// TwinCAT 3 PLC project Controller
// Title: BIO2
// Company: 3P Innovation Ltd.
// Author: James Tyler
// ProgramVersion: 3.1.0.8
// libraries:
//   Standard, * (System)
//   Tc2_Standard, * (Beckhoff Automation GmbH)
//   Tc2_System, * (Beckhoff Automation GmbH)
//   Tc2_Utilities, * (Beckhoff Automation GmbH)
//   Tc2_XmlDataSrv, * (Beckhoff Automation GmbH)
//   Tc3_Interfaces, * (Beckhoff Automation GmbH)
//   Tc3_Module, * (Beckhoff Automation GmbH)
//   Tc_Persistent, * (Red Rock Controls Limited)
//   Tc2_MC2,newest,Beckhoff Automation GmbH
//   Tc_Collections,1.0.0.8,Red Rock Controls
//   Tc_Helper,1.0.0.8,Red Rock Controls
// project tree:
//   Classes/Compress/ FB_Compress.TcPOU
//   Classes/Config/ TConfig.TcPOU, TConfigData.TcDUT
//   Classes/Pusher/ FB_Pusher.TcPOU
//   Classes/Shield/ FB_Shield.TcPOU
//   DUTs/ st_language.TcDUT, St_Compress_Settings.TcDUT, E_LampState.TcDUT, E_CTRL_STATE.TcDUT (not stored), st_graph_visibility.TcDUT, Limits.TcDUT, Recipe.TcDUT (not stored), Rec_Compress.TcDUT, Rec_Other.TcDUT, Rec_Pusher.TcDUT, Rec_Clamp.TcDUT, Rec_Shield.TcDUT, st_recipe_titles.TcDUT, st_yellow_visibility.TcDUT
//   GVLs/ GVL_IO.TcGVL, GVL_Objects.TcGVL, GVL_ZenOn.TcGVL
//   / PlcTask.TcTTO, Task_Fast.TcTTO
//   POUs/ Config_Slow.TcPOU, FB_AxisControl.TcPOU, FB_LampController.TcPOU (not stored), F_DisplayText.TcPOU, PRG_MAIN.TcPOU, PRG_IO.TcPOU, PRG_Machine.TcPOU
//   XML/ eXMLState.TcDUT (not stored), FB_Retain.TcPOU (not stored), FB_RetainedData.TcPOU
// real-time tasks:
//   TASK PlcTask: cycle T#10ms, priority 12, ADS port 350
//   TASK Task_Fast: cycle T#1ms, priority 4, ADS port 351
// motion (NC):
//   TASK NC-Task 1 SAF: cycle T#2ms, priority 6, ADS port 501
//   TASK NC-Task 1 SVB: cycle T#10ms, priority 10, ADS port 511
//   AXIS Compress (id 1)
//     Dynamic: Acceleration=60.7875, Deceleration=60.7875, Jerk=182.363
//     Velo: RefSearch=0.40525, RefSync=0.40525, SlowManual=2.02625, FastManual=12.1575, Fast=40.525, Maximum=200
//     OtherSettings: AllowMotionCmdToSlave=true
//     encoder EncType=19
//       EncPara: ScaleFactorNumerator=0.5, ScaleFactorDenominator=1048576, ModuloFactor=0.5, MaxCount=#xffffffff
//     drive DrvType=16
//       DrvPara: MaxCount=#xffffffff
//         Analog: VeloReferenz=200, VeloScale=32
//         TimeComp: TaskDelayCycles=1
//     controller CtrType=1
//       CtrPara: PriorControlFactor=1
//         PosDiffControl: Enable=false, Range=0.05
//         PID: PosKp=20
//         Observer: BandWidth=20
//   AXIS Pusher (id 2)
//     Dynamic: Acceleration=60.7875, Deceleration=60.7875, Jerk=182.363
//     Velo: RefSearch=0.40525, RefSync=0.40525, SlowManual=2.02625, FastManual=12.1575, Fast=40.525, Maximum=40.525
//     OtherSettings: AllowMotionCmdToSlave=true
//     encoder EncType=19
//       EncPara: ScaleFactorNumerator=0.5, ScaleFactorDenominator=1048576, ModuloFactor=0.5, MaxCount=#xffffffff
//     drive DrvType=16
//       DrvPara: MaxCount=#xffffffff
//         Analog: VeloReferenz=100, VeloScale=32
//         TimeComp: TaskDelayCycles=1
//     controller CtrType=1
//       CtrPara: PriorControlFactor=1
//         PosDiffControl: Enable=false, Range=0.5
//         PID: PosKp=20
//         Observer: BandWidth=20
//   AXIS Shield (id 3)
//     Dynamic: Acceleration=60.7875, Deceleration=60.7875, Jerk=182.363
//     Velo: RefSearch=0.40525, RefSync=0.40525, SlowManual=2.02625, FastManual=12.1575, Fast=200, Maximum=200
//     OtherSettings: AllowMotionCmdToSlave=true
//     encoder EncType=19
//       EncPara: ScaleFactorNumerator=0.5, ScaleFactorDenominator=1048576, ModuloFactor=0.5, MaxCount=#xffffffff
//     drive DrvType=16
//       DrvPara: MaxCount=#xffffffff
//         Analog: VeloReferenz=200, VeloScale=32
//         TimeComp: TaskDelayCycles=1
//     controller CtrType=1
//       CtrPara: PriorControlFactor=1
//         PosDiffControl: Enable=false, Range=0.05
//         PID: PosKp=20
//         Observer: BandWidth=20
// I/O:
//   DEVICE Device 1 (EtherCAT), AmsNetId 5.49.191.228.2.1
//     Term 5 (EK1100) [EK1100 EtherCAT Coupler (2A E-Bus)]
//       Term 6 (EL1809) [EL1809 16Ch. Dig. Input 24V, 3ms]
//       Term 7 (EL2798) [EL2798 8Ch. Dig. Output 24V AC/DC, 2A, potential-free]
//       Term 13 (EL9011) [EL9011 End Terminal]
//     Term 8 (EK1100) [EK1100 EtherCAT Coupler (2A E-Bus)]
//       Term 9 (EL7201-9014) [EL7201-9014 1Ch. MDP742 Servo motor output stage with OCT (50V, 4A) and STO input]
//       Term 10 (EL7201-9014) [EL7201-9014 1Ch. MDP742 Servo motor output stage with OCT (50V, 4A)  and STO input]
//       Term 11 (EL7201-9014) [EL7201-9014 1Ch. MDP742 Servo motor output stage with OCT (50V, 4A)  and STO input]
//       Term 12 (EL1809) [EL1809 16Ch. Dig. Input 24V, 3ms]
//       Term 14 (EL9011) [EL9011 End Terminal]
//   DEVICE Device 3 (RT-Ethernet Protocol) (disabled), AmsNetId 5.49.191.228.4.1
// variable links:
//   NC-Task 1 SAF/Axes/Compress <-> Device 1 (EtherCAT)/Term 8 (EK1100)/Term 9 (EL7201-9014)
//     Drive/Inputs/In/nDcOutputTime <-> InfoData/DcOutputShift
//     Drive/Inputs/In/nState1 <-> DRV Statusword/Statusword
//     Drive/Inputs/In/nState2 <-> DRV Statusword/Statusword @bit 8
//     Drive/Inputs/In/nState4 @bit 1 <-> WcState/InputToggle
//     Drive/Inputs/In/nState4 <-> WcState/WcState
//     Drive/Outputs/Out/nCtrl1 <-> DRV Controlword/Controlword
//     Drive/Outputs/Out/nCtrl2 <-> DRV Controlword/Controlword @bit 8
//     Drive/Outputs/Out/nDataOut2 <-> DRV Target velocity/Target velocity
//     Enc/Inputs/In/nDataIn1 <-> FB Position/Position
//     Enc/Inputs/In/nDcInputTime <-> InfoData/DcInputShift
//     Enc/Inputs/In/nState4 @bit 1 <-> WcState/InputToggle
//     Enc/Inputs/In/nState4 <-> WcState/WcState
//   NC-Task 1 SAF/Axes/Pusher <-> Device 1 (EtherCAT)/Term 8 (EK1100)/Term 10 (EL7201-9014)
//     Drive/Inputs/In/nDcOutputTime <-> InfoData/DcOutputShift
//     Drive/Inputs/In/nState1 <-> DRV Statusword/Statusword
//     Drive/Inputs/In/nState2 <-> DRV Statusword/Statusword @bit 8
//     Drive/Inputs/In/nState4 @bit 1 <-> WcState/InputToggle
//     Drive/Inputs/In/nState4 <-> WcState/WcState
//     Drive/Outputs/Out/nCtrl1 <-> DRV Controlword/Controlword
//     Drive/Outputs/Out/nCtrl2 <-> DRV Controlword/Controlword @bit 8
//     Drive/Outputs/Out/nDataOut2 <-> DRV Target velocity/Target velocity
//     Enc/Inputs/In/nDataIn1 <-> FB Position/Position
//     Enc/Inputs/In/nDcInputTime <-> InfoData/DcInputShift
//     Enc/Inputs/In/nState4 @bit 1 <-> WcState/InputToggle
//     Enc/Inputs/In/nState4 <-> WcState/WcState
//   NC-Task 1 SAF/Axes/Shield <-> Device 1 (EtherCAT)/Term 8 (EK1100)/Term 11 (EL7201-9014)
//     Drive/Inputs/In/nDcOutputTime <-> InfoData/DcOutputShift
//     Drive/Inputs/In/nState1 <-> DRV Statusword/Statusword
//     Drive/Inputs/In/nState2 <-> DRV Statusword/Statusword @bit 8
//     Drive/Inputs/In/nState4 @bit 1 <-> WcState/InputToggle
//     Drive/Inputs/In/nState4 <-> WcState/WcState
//     Drive/Outputs/Out/nCtrl1 <-> DRV Controlword/Controlword
//     Drive/Outputs/Out/nCtrl2 <-> DRV Controlword/Controlword @bit 8
//     Drive/Outputs/Out/nDataOut2 <-> DRV Target velocity/Target velocity
//     Enc/Inputs/In/nDataIn1 <-> FB Position/Position
//     Enc/Inputs/In/nDcInputTime <-> InfoData/DcInputShift
//     Enc/Inputs/In/nState4 @bit 1 <-> WcState/InputToggle
//     Enc/Inputs/In/nState4 <-> WcState/WcState
//   Controller/Controller Instance <-> Device 1 (EtherCAT)/Term 5 (EK1100)/Term 6 (EL1809)
//     PlcTask Inputs/GVL_IO.ixCabinetE_StopButtonOkay <-> Channel 1/Cabinet E-Stop
//     PlcTask Inputs/GVL_IO.ixE_StopRelayOkay <-> Channel 2/Input
//     PlcTask Inputs/GVL_IO.ixGuardRelayOkay <-> Channel 3/Input
//     PlcTask Inputs/GVL_IO.ixResetButton <-> Channel 6/Input
//     PlcTask Inputs/GVL_IO.ixSpareIN4 <-> Channel 4/Input
//     PlcTask Inputs/GVL_IO.ixSpareIN5 <-> Channel 5/Input
//     PlcTask Inputs/GVL_IO.ixSpareIN7 <-> Channel 7/Input
//     PlcTask Inputs/GVL_IO.ixSpareIN8 <-> Channel 8/Input
//     PlcTask Inputs/GVL_IO.ixStartButton <-> Channel 9/Input
//     PlcTask Inputs/GVL_IO.ixStop_Button <-> Channel 10/Input
//   Controller/Controller Instance <-> Device 1 (EtherCAT)/Term 5 (EK1100)/Term 7 (EL2798)
//     PlcTask Outputs/GVL_IO.qxClamp <-> Channel 2/Output
//     PlcTask Outputs/GVL_IO.qxEnableE_Stop <-> Channel 1/Output
//     PlcTask Outputs/GVL_IO.qxResetButtonLamp <-> Channel 5/Output
//     PlcTask Outputs/GVL_IO.qxSpareOUT3 <-> Channel 3/Output
//     PlcTask Outputs/GVL_IO.qxStartButtonLamp <-> Channel 4/Output
//   Controller/Controller Instance <-> Device 1 (EtherCAT)/Term 8 (EK1100)/Term 10 (EL7201-9014)
//     PlcTask Inputs/GVL_IO.ibPusherServoTorque <-> DRV Torque actual value/Torque actual value
//   Controller/Controller Instance <-> Device 1 (EtherCAT)/Term 8 (EK1100)/Term 11 (EL7201-9014)
//     PlcTask Inputs/GVL_IO.ibShieldServoTorque <-> DRV Torque actual value/Torque actual value
//   Controller/Controller Instance <-> Device 1 (EtherCAT)/Term 8 (EK1100)/Term 12 (EL1809)
//     PlcTask Inputs/GVL_IO.ixCompressHomeSwitch <-> Channel 1/Input
//     PlcTask Inputs/GVL_IO.ixFanCartridgeDiagnostics <-> Channel 11/Input
//     PlcTask Inputs/GVL_IO.ixGuardOkay <-> Channel 9/Input
//     PlcTask Inputs/GVL_IO.ixMachineE_StopButtonOkay <-> Channel 10/Input
//     PlcTask Inputs/GVL_IO.ixPusherHomeSwitch <-> Channel 3/Input
//     PlcTask Inputs/GVL_IO.ixShieldHomeSwitch <-> Channel 5/Input
//     PlcTask Inputs/GVL_IO.ixStart_Button_Machine <-> Channel 7/Input
//   Controller/Controller Instance <-> Device 1 (EtherCAT)/Term 8 (EK1100)/Term 9 (EL7201-9014)
//     PlcTask Inputs/GVL_IO.ibCompressServoTorque <-> DRV Torque actual value/Torque actual value
//   Controller/Controller Instance <-> NC-Task 1 SAF/Axes/Compress
//     PlcTask Inputs/GVL_IO.CompressAxis.NcToPlc <-> Outputs/ToPlc
//     PlcTask Outputs/GVL_IO.CompressAxis.PlcToNc <-> Inputs/FromPlc
//   Controller/Controller Instance <-> NC-Task 1 SAF/Axes/Pusher
//     PlcTask Inputs/GVL_IO.PusherAxis.NcToPlc <-> Outputs/ToPlc
//     PlcTask Outputs/GVL_IO.PusherAxis.PlcToNc <-> Inputs/FromPlc
//   Controller/Controller Instance <-> NC-Task 1 SAF/Axes/Shield
//     PlcTask Inputs/GVL_IO.ShieldAxis.NcToPlc <-> Outputs/ToPlc
//     PlcTask Outputs/GVL_IO.ShieldAxis.PlcToNc <-> Inputs/FromPlc

CONFIGURATION Controller
    RESOURCE PLC ON TwinCAT3
        TASK PlcTask(INTERVAL := T#10ms, PRIORITY := 12);
        TASK Task_Fast(INTERVAL := T#1ms, PRIORITY := 4);
        PROGRAM PRG_MAIN WITH PlcTask : PRG_MAIN;
        PROGRAM Config_Slow WITH Task_Fast : Config_Slow;
    END_RESOURCE
END_CONFIGURATION

// ---- Classes/Config/TConfigData.TcDUT
{attribute 'pack_mode' := '0'}
TYPE TConfigData :
STRUCT
	
	//Limits
	con_max_limit_Compress 					:LREAL;
	con_max_limit_Shield 					:LREAL;
	con_max_limit_Pusher 					:LREAL;
	con_max_pusher_shield_diff				:LREAL;
	con_max_torque							:LREAL;
	
	//you are here
	//Rec1_Name        						:STRING;
	rec1_Name_1									:UDINT;
	rec1_Name_2									:UDINT;
	rec1_Name_3									:UDINT;
	rec1_Name_4									:UDINT;
	rec1_Name_5									:UDINT;
	
	rec1_Shield_Retract_Speed					:LREAL;
	rec1_Shield_Speed_1							:LREAL;
	rec1_Shield_Speed_2							:LREAL;
	rec1_Shield_Speed_3							:LREAL;
	rec1_Shield_Speed_4							:LREAL;
	rec1_Shield_Speed_5							:LREAL;
	rec1_Shield_Speed_6							:LREAL;
	rec1_Shield_Distance_1						:LREAL;
	rec1_Shield_Distance_2						:LREAL;
	rec1_Shield_Distance_3						:LREAL;
	rec1_shield_Distance_4						:LREAL;
	rec1_shield_Distance_5						:LREAL;
	rec1_shield_Distance_6						:LREAL;
	
	rec1_Compress_Initial_Speed					:LREAL;
	rec1_Compress_Initial_Distance				:LREAL;
	rec1_Compress_Relax_Distance					:LREAL;
	rec1_Compress_Retract_Speed					:LREAL;
	
	rec1_Pusher_Retract_Speed					:LREAL;
	rec1_Pusher_Speed_1							:LREAL;
	rec1_Pusher_Speed_2							:LREAL;
	rec1_Pusher_Speed_3							:LREAL;
	rec1_Pusher_Speed_4							:LREAL;
	rec1_Pusher_Speed_5							:LREAL;
	rec1_Pusher_Speed_6							:LREAL;
	rec1_Pusher_Distance_1						:LREAL;
	rec1_Pusher_Distance_2						:LREAL;
	rec1_Pusher_Distance_3						:LREAL;
	rec1_Pusher_Distance_4						:LREAL;
	rec1_Pusher_Distance_5						:LREAL;
	rec1_Pusher_Distance_6						:LREAL;
	
	rec1_Other_Compress_Home_Offset				:LREAL;
	rec1_Other_Pusher_Home_Offset				:LREAL;
	rec1_Other_Shield_Home_Offset				:LREAL;
	
	rec1_Clamp_Release_Instance					:LREAL;
	
	rec1_Memory_Free							:LREAL:=1;

	//Rec2_Name        						:STRING;
	rec2_Name_1									:UDINT;
	rec2_Name_2									:UDINT;
	rec2_Name_3									:UDINT;
	rec2_Name_4									:UDINT;
	rec2_Name_5									:UDINT;
	
	rec2_Shield_Retract_Speed					:LREAL;
	rec2_Shield_Speed_1							:LREAL;
	rec2_Shield_Speed_2							:LREAL;
	rec2_Shield_Speed_3							:LREAL;
	rec2_Shield_Speed_4							:LREAL;
	rec2_Shield_Speed_5							:LREAL;
	rec2_Shield_Speed_6							:LREAL;
	rec2_Shield_Distance_1						:LREAL;
	rec2_Shield_Distance_2						:LREAL;
	rec2_Shield_Distance_3						:LREAL;
	rec2_shield_Distance_4						:LREAL;
	rec2_shield_Distance_5						:LREAL;
	rec2_shield_Distance_6						:LREAL;
	
	rec2_Compress_Initial_Speed					:LREAL;
	rec2_Compress_Initial_Distance				:LREAL;
	rec2_Compress_Relax_Distance					:LREAL;
	rec2_Compress_Retract_Speed					:LREAL;
	
	rec2_Pusher_Retract_Speed					:LREAL;
	rec2_Pusher_Speed_1							:LREAL;
	rec2_Pusher_Speed_2							:LREAL;
	rec2_Pusher_Speed_3							:LREAL;
	rec2_Pusher_Speed_4							:LREAL;
	rec2_Pusher_Speed_5							:LREAL;
	rec2_Pusher_Speed_6							:LREAL;
	rec2_Pusher_Distance_1						:LREAL;
	rec2_Pusher_Distance_2						:LREAL;
	rec2_Pusher_Distance_3						:LREAL;
	rec2_Pusher_Distance_4						:LREAL;
	rec2_Pusher_Distance_5						:LREAL;
	rec2_Pusher_Distance_6						:LREAL;
	
	rec2_Other_Compress_Home_Offset				:LREAL;
	rec2_Other_Pusher_Home_Offset				:LREAL;
	rec2_Other_Shield_Home_Offset				:LREAL;
	
	rec2_Clamp_Release_Instance					:LREAL;
	
	rec2_Memory_Free							:LREAL:=1;

	//Rec3_Name        						:STRING;
	rec3_Name_1									:UDINT;
	rec3_Name_2									:UDINT;
	rec3_Name_3									:UDINT;
	rec3_Name_4									:UDINT;
	rec3_Name_5									:UDINT;
	
	rec3_Shield_Retract_Speed					:LREAL;
	rec3_Shield_Speed_1							:LREAL;
	rec3_Shield_Speed_2							:LREAL;
	rec3_Shield_Speed_3							:LREAL;
	rec3_Shield_Speed_4							:LREAL;
	rec3_Shield_Speed_5							:LREAL;
	rec3_Shield_Speed_6							:LREAL;
	rec3_Shield_Distance_1						:LREAL;
	rec3_Shield_Distance_2						:LREAL;
	rec3_Shield_Distance_3						:LREAL;
	rec3_shield_Distance_4						:LREAL;
	rec3_shield_Distance_5						:LREAL;
	rec3_shield_Distance_6						:LREAL;
	
	rec3_Compress_Initial_Speed					:LREAL;
	rec3_Compress_Initial_Distance				:LREAL;
	rec3_Compress_Relax_Distance					:LREAL;
	rec3_Compress_Retract_Speed					:LREAL;
	
	rec3_Pusher_Retract_Speed					:LREAL;
	rec3_Pusher_Speed_1							:LREAL;
	rec3_Pusher_Speed_2							:LREAL;
	rec3_Pusher_Speed_3							:LREAL;
	rec3_Pusher_Speed_4							:LREAL;
	rec3_Pusher_Speed_5							:LREAL;
	rec3_Pusher_Speed_6							:LREAL;
	rec3_Pusher_Distance_1						:LREAL;
	rec3_Pusher_Distance_2						:LREAL;
	rec3_Pusher_Distance_3						:LREAL;
	rec3_Pusher_Distance_4						:LREAL;
	rec3_Pusher_Distance_5						:LREAL;
	rec3_Pusher_Distance_6						:LREAL;
	
	rec3_Other_Compress_Home_Offset				:LREAL;
	rec3_Other_Pusher_Home_Offset				:LREAL;
	rec3_Other_Shield_Home_Offset				:LREAL;
	
	rec3_Clamp_Release_Instance					:LREAL;
	
	rec3_Memory_Free							:LREAL:=1;

	//Rec4_Name        						:STRING;
	rec4_Name_1									:UDINT;
	rec4_Name_2									:UDINT;
	rec4_Name_3									:UDINT;
	rec4_Name_4									:UDINT;
	rec4_Name_5									:UDINT;
	
	rec4_Shield_Retract_Speed					:LREAL;
	rec4_Shield_Speed_1							:LREAL;
	rec4_Shield_Speed_2							:LREAL;
	rec4_Shield_Speed_3							:LREAL;
	rec4_Shield_Speed_4							:LREAL;
	rec4_Shield_Speed_5							:LREAL;
	rec4_Shield_Speed_6							:LREAL;
	rec4_Shield_Distance_1						:LREAL;
	rec4_Shield_Distance_2						:LREAL;
	rec4_Shield_Distance_3						:LREAL;
	rec4_shield_Distance_4						:LREAL;
	rec4_shield_Distance_5						:LREAL;
	rec4_shield_Distance_6						:LREAL;
	
	rec4_Compress_Initial_Speed					:LREAL;
	rec4_Compress_Initial_Distance				:LREAL;
	rec4_Compress_Relax_Distance					:LREAL;
	rec4_Compress_Retract_Speed					:LREAL;
	
	rec4_Pusher_Retract_Speed					:LREAL;
	rec4_Pusher_Speed_1							:LREAL;
	rec4_Pusher_Speed_2							:LREAL;
	rec4_Pusher_Speed_3							:LREAL;
	rec4_Pusher_Speed_4							:LREAL;
	rec4_Pusher_Speed_5							:LREAL;
	rec4_Pusher_Speed_6							:LREAL;
	rec4_Pusher_Distance_1						:LREAL;
	rec4_Pusher_Distance_2						:LREAL;
	rec4_Pusher_Distance_3						:LREAL;
	rec4_Pusher_Distance_4						:LREAL;
	rec4_Pusher_Distance_5						:LREAL;
	rec4_Pusher_Distance_6						:LREAL;
	
	rec4_Other_Compress_Home_Offset				:LREAL;
	rec4_Other_Pusher_Home_Offset				:LREAL;
	rec4_Other_Shield_Home_Offset				:LREAL;
	
	rec4_Clamp_Release_Instance					:LREAL;

	rec4_Memory_Free							:LREAL:=1;		
	
	//Rec5_Name        						:STRING;
	rec5_Name_1									:UDINT;
	rec5_Name_2									:UDINT;
	rec5_Name_3									:UDINT;
	rec5_Name_4									:UDINT;
	rec5_Name_5									:UDINT;
	
	rec5_Shield_Retract_Speed					:LREAL;
	rec5_Shield_Speed_1							:LREAL;
	rec5_Shield_Speed_2							:LREAL;
	rec5_Shield_Speed_3							:LREAL;
	rec5_Shield_Speed_4							:LREAL;
	rec5_Shield_Speed_5							:LREAL;
	rec5_Shield_Speed_6							:LREAL;
	rec5_Shield_Distance_1						:LREAL;
	rec5_Shield_Distance_2						:LREAL;
	rec5_Shield_Distance_3						:LREAL;
	rec5_shield_Distance_4						:LREAL;
	rec5_shield_Distance_5						:LREAL;
	rec5_shield_Distance_6						:LREAL;
	
	rec5_Compress_Initial_Speed					:LREAL;
	rec5_Compress_Initial_Distance				:LREAL;
	rec5_Compress_Relax_Distance					:LREAL;
	rec5_Compress_Retract_Speed					:LREAL;
	
	rec5_Pusher_Retract_Speed					:LREAL;
	rec5_Pusher_Speed_1							:LREAL;
	rec5_Pusher_Speed_2							:LREAL;
	rec5_Pusher_Speed_3							:LREAL;
	rec5_Pusher_Speed_4							:LREAL;
	rec5_Pusher_Speed_5							:LREAL;
	rec5_Pusher_Speed_6							:LREAL;
	rec5_Pusher_Distance_1						:LREAL;
	rec5_Pusher_Distance_2						:LREAL;
	rec5_Pusher_Distance_3						:LREAL;
	rec5_Pusher_Distance_4						:LREAL;
	rec5_Pusher_Distance_5						:LREAL;
	rec5_Pusher_Distance_6						:LREAL;
	
	rec5_Other_Compress_Home_Offset				:LREAL;
	rec5_Other_Pusher_Home_Offset				:LREAL;
	rec5_Other_Shield_Home_Offset				:LREAL;
	
	rec5_Clamp_Release_Instance					:LREAL;
	
	rec5_Memory_Free							:LREAL:=1;
	
	//Rec6_Name        						:STRING;
	rec6_Name_1									:UDINT;
	rec6_Name_2									:UDINT;
	rec6_Name_3									:UDINT;
	rec6_Name_4									:UDINT;
	rec6_Name_5									:UDINT;
	
	rec6_Shield_Retract_Speed					:LREAL;
	rec6_Shield_Speed_1							:LREAL;
	rec6_Shield_Speed_2							:LREAL;
	rec6_Shield_Speed_3							:LREAL;
	rec6_Shield_Speed_4							:LREAL;
	rec6_Shield_Speed_5							:LREAL;
	rec6_Shield_Speed_6							:LREAL;
	rec6_Shield_Distance_1						:LREAL;
	rec6_Shield_Distance_2						:LREAL;
	rec6_Shield_Distance_3						:LREAL;
	rec6_shield_Distance_4						:LREAL;
	rec6_shield_Distance_5						:LREAL;
	rec6_shield_Distance_6						:LREAL;
	
	rec6_Compress_Initial_Speed					:LREAL;
	rec6_Compress_Initial_Distance				:LREAL;
	rec6_Compress_Relax_Distance					:LREAL;
	rec6_Compress_Retract_Speed					:LREAL;
	
	rec6_Pusher_Retract_Speed					:LREAL;
	rec6_Pusher_Speed_1							:LREAL;
	rec6_Pusher_Speed_2							:LREAL;
	rec6_Pusher_Speed_3							:LREAL;
	rec6_Pusher_Speed_4							:LREAL;
	rec6_Pusher_Speed_5							:LREAL;
	rec6_Pusher_Speed_6							:LREAL;
	rec6_Pusher_Distance_1						:LREAL;
	rec6_Pusher_Distance_2						:LREAL;
	rec6_Pusher_Distance_3						:LREAL;
	rec6_Pusher_Distance_4						:LREAL;
	rec6_Pusher_Distance_5						:LREAL;
	rec6_Pusher_Distance_6						:LREAL;
	
	rec6_Other_Compress_Home_Offset				:LREAL;
	rec6_Other_Pusher_Home_Offset				:LREAL;
	rec6_Other_Shield_Home_Offset				:LREAL;
	
	rec6_Clamp_Release_Instance					:LREAL;
	
	rec6_Memory_Free							:LREAL:=1;
	
	//Rec7_Name        						:STRING;
	rec7_Name_1									:UDINT;
	rec7_Name_2									:UDINT;
	rec7_Name_3									:UDINT;
	rec7_Name_4									:UDINT;
	rec7_Name_5									:UDINT;
	
	rec7_Shield_Retract_Speed					:LREAL;
	rec7_Shield_Speed_1							:LREAL;
	rec7_Shield_Speed_2							:LREAL;
	rec7_Shield_Speed_3							:LREAL;
	rec7_Shield_Speed_4							:LREAL;
	rec7_Shield_Speed_5							:LREAL;
	rec7_Shield_Speed_6							:LREAL;
	rec7_Shield_Distance_1						:LREAL;
	rec7_Shield_Distance_2						:LREAL;
	rec7_Shield_Distance_3						:LREAL;
	rec7_shield_Distance_4						:LREAL;
	rec7_shield_Distance_5						:LREAL;
	rec7_shield_Distance_6						:LREAL;
	
	rec7_Compress_Initial_Speed					:LREAL;
	rec7_Compress_Initial_Distance				:LREAL;
	rec7_Compress_Relax_Distance					:LREAL;
	rec7_Compress_Retract_Speed					:LREAL;
	
	rec7_Pusher_Retract_Speed					:LREAL;
	rec7_Pusher_Speed_1							:LREAL;
	rec7_Pusher_Speed_2							:LREAL;
	rec7_Pusher_Speed_3							:LREAL;
	rec7_Pusher_Speed_4							:LREAL;
	rec7_Pusher_Speed_5							:LREAL;
	rec7_Pusher_Speed_6							:LREAL;
	rec7_Pusher_Distance_1						:LREAL;
	rec7_Pusher_Distance_2						:LREAL;
	rec7_Pusher_Distance_3						:LREAL;
	rec7_Pusher_Distance_4						:LREAL;
	rec7_Pusher_Distance_5						:LREAL;
	rec7_Pusher_Distance_6						:LREAL;
	
	rec7_Other_Compress_Home_Offset				:LREAL;
	rec7_Other_Pusher_Home_Offset				:LREAL;
	rec7_Other_Shield_Home_Offset				:LREAL;
	
	rec7_Clamp_Release_Instance					:LREAL;
	
	rec7_Memory_Free							:LREAL:=1;
	
	//Rec8_Name        						:STRING;
	rec8_Name_1									:UDINT;
	rec8_Name_2									:UDINT;
	rec8_Name_3									:UDINT;
	rec8_Name_4									:UDINT;
	rec8_Name_5									:UDINT;
	
	rec8_Shield_Retract_Speed					:LREAL;
	rec8_Shield_Speed_1							:LREAL;
	rec8_Shield_Speed_2							:LREAL;
	rec8_Shield_Speed_3							:LREAL;
	rec8_Shield_Speed_4							:LREAL;
	rec8_Shield_Speed_5							:LREAL;
	rec8_Shield_Speed_6							:LREAL;
	rec8_Shield_Distance_1						:LREAL;
	rec8_Shield_Distance_2						:LREAL;
	rec8_Shield_Distance_3						:LREAL;
	rec8_shield_Distance_4						:LREAL;
	rec8_shield_Distance_5						:LREAL;
	rec8_shield_Distance_6						:LREAL;
	
	rec8_Compress_Initial_Speed					:LREAL;
	rec8_Compress_Initial_Distance				:LREAL;
	rec8_Compress_Relax_Distance					:LREAL;
	rec8_Compress_Retract_Speed					:LREAL;
	
	rec8_Pusher_Retract_Speed					:LREAL;
	rec8_Pusher_Speed_1							:LREAL;
	rec8_Pusher_Speed_2							:LREAL;
	rec8_Pusher_Speed_3							:LREAL;
	rec8_Pusher_Speed_4							:LREAL;
	rec8_Pusher_Speed_5							:LREAL;
	rec8_Pusher_Speed_6							:LREAL;
	rec8_Pusher_Distance_1						:LREAL;
	rec8_Pusher_Distance_2						:LREAL;
	rec8_Pusher_Distance_3						:LREAL;
	rec8_Pusher_Distance_4						:LREAL;
	rec8_Pusher_Distance_5						:LREAL;
	rec8_Pusher_Distance_6						:LREAL;
	
	rec8_Other_Compress_Home_Offset				:LREAL;
	rec8_Other_Pusher_Home_Offset				:LREAL;
	rec8_Other_Shield_Home_Offset				:LREAL;
	
	rec8_Clamp_Release_Instance					:LREAL;
	
	rec8_Memory_Free							:LREAL:=1;
	
	//Rec9_Name        						:STRING;
	rec9_Name_1									:UDINT;
	rec9_Name_2									:UDINT;
	rec9_Name_3									:UDINT;
	rec9_Name_4									:UDINT;
	rec9_Name_5									:UDINT;
	
	rec9_Shield_Retract_Speed					:LREAL;
	rec9_Shield_Speed_1							:LREAL;
	rec9_Shield_Speed_2							:LREAL;
	rec9_Shield_Speed_3							:LREAL;
	rec9_Shield_Speed_4							:LREAL;
	rec9_Shield_Speed_5							:LREAL;
	rec9_Shield_Speed_6							:LREAL;
	rec9_Shield_Distance_1						:LREAL;
	rec9_Shield_Distance_2						:LREAL;
	rec9_Shield_Distance_3						:LREAL;
	rec9_shield_Distance_4						:LREAL;
	rec9_shield_Distance_5						:LREAL;
	rec9_shield_Distance_6						:LREAL;
	
	rec9_Compress_Initial_Speed					:LREAL;
	rec9_Compress_Initial_Distance				:LREAL;
	rec9_Compress_Relax_Distance					:LREAL;
	rec9_Compress_Retract_Speed					:LREAL;
	
	rec9_Pusher_Retract_Speed					:LREAL;
	rec9_Pusher_Speed_1							:LREAL;
	rec9_Pusher_Speed_2							:LREAL;
	rec9_Pusher_Speed_3							:LREAL;
	rec9_Pusher_Speed_4							:LREAL;
	rec9_Pusher_Speed_5							:LREAL;
	rec9_Pusher_Speed_6							:LREAL;
	rec9_Pusher_Distance_1						:LREAL;
	rec9_Pusher_Distance_2						:LREAL;
	rec9_Pusher_Distance_3						:LREAL;
	rec9_Pusher_Distance_4						:LREAL;
	rec9_Pusher_Distance_5						:LREAL;
	rec9_Pusher_Distance_6						:LREAL;
	
	rec9_Other_Compress_Home_Offset				:LREAL;
	rec9_Other_Pusher_Home_Offset				:LREAL;
	rec9_Other_Shield_Home_Offset				:LREAL;
	
	rec9_Clamp_Release_Instance					:LREAL;
	
	rec9_Memory_Free							:LREAL:=1;
	
	//Rec10_Name        						:STRING;
	rec10_Name_1									:UDINT;
	rec10_Name_2									:UDINT;
	rec10_Name_3									:UDINT;
	rec10_Name_4									:UDINT;
	rec10_Name_5									:UDINT;
	
	rec10_Shield_Retract_Speed					:LREAL;
	rec10_Shield_Speed_1							:LREAL;
	rec10_Shield_Speed_2							:LREAL;
	rec10_Shield_Speed_3							:LREAL;
	rec10_Shield_Speed_4							:LREAL;
	rec10_Shield_Speed_5							:LREAL;
	rec10_Shield_Speed_6							:LREAL;
	rec10_Shield_Distance_1						:LREAL;
	rec10_Shield_Distance_2						:LREAL;
	rec10_Shield_Distance_3						:LREAL;
	rec10_shield_Distance_4						:LREAL;
	rec10_shield_Distance_5						:LREAL;
	rec10_shield_Distance_6						:LREAL;
	
	rec10_Compress_Initial_Speed					:LREAL;
	rec10_Compress_Initial_Distance				:LREAL;
	rec10_Compress_Relax_Distance					:LREAL;
	rec10_Compress_Retract_Speed					:LREAL;
	
	rec10_Pusher_Retract_Speed					:LREAL;
	rec10_Pusher_Speed_1							:LREAL;
	rec10_Pusher_Speed_2							:LREAL;
	rec10_Pusher_Speed_3							:LREAL;
	rec10_Pusher_Speed_4							:LREAL;
	rec10_Pusher_Speed_5							:LREAL;
	rec10_Pusher_Speed_6							:LREAL;
	rec10_Pusher_Distance_1						:LREAL;
	rec10_Pusher_Distance_2						:LREAL;
	rec10_Pusher_Distance_3						:LREAL;
	rec10_Pusher_Distance_4						:LREAL;
	rec10_Pusher_Distance_5						:LREAL;
	rec10_Pusher_Distance_6						:LREAL;
	
	rec10_Other_Compress_Home_Offset				:LREAL;
	rec10_Other_Pusher_Home_Offset				:LREAL;
	rec10_Other_Shield_Home_Offset				:LREAL;
	
	rec10_Clamp_Release_Instance					:LREAL;

	rec10_Memory_Free							:LREAL:=1;	
	
	(*Initialised - MUST BE LAST VARIABLE IN STUCTURE*)
    Initialised : BOOL;
END_STRUCT
END_TYPE

// ---- DUTs/st_language.TcDUT
TYPE st_language :
STRUCT
	portuguese				:BOOL:=FALSE;
	english					:BOOL:=TRUE;
END_STRUCT
END_TYPE

// ---- DUTs/St_Compress_Settings.TcDUT
TYPE St_Compress_Settings :
STRUCT
	
	//compress setting
	button					:BOOL;
	plus					:BOOL;
	minus					:BOOL;
	find					:BOOL;
	speed					:LREAL:=2;
	distance				:LREAL;
	old_distance			:LREAL;
	distance_vis			:BOOL;
	done					:BOOL;
	
END_STRUCT
END_TYPE

// ---- DUTs/E_LampState.TcDUT
TYPE E_LampState : 
(
	Off := 0,
    Steady := 1,
    FastFlash := 2,
    SlowFlash := 4
);
END_TYPE

// ---- DUTs/st_graph_visibility.TcDUT
TYPE st_graph_visibility :
	STRUCT
		shield_speed_1						:BOOL;
		shield_speed_2						:BOOL;
		shield_speed_3						:BOOL;
		shield_speed_4						:BOOL;
		shield_speed_5						:BOOL;
		shield_speed_6						:BOOL;
		shield_distance_1					:BOOL;
		shield_distance_2					:BOOL;
		shield_distance_3					:BOOL;
		shield_distance_4					:BOOL;
		shield_distance_5					:BOOL;
		shield_distance_6					:BOOL;
		shield_retract						:BOOL;
		
		pusher_speed_1						:BOOL;
		pusher_speed_2						:BOOL;
		pusher_speed_3						:BOOL;
		pusher_speed_4						:BOOL;
		pusher_speed_5						:BOOL;
		pusher_speed_6						:BOOL;
		pusher_distance_1					:BOOL;
		pusher_distance_2					:BOOL;
		pusher_distance_3					:BOOL;
		pusher_distance_4					:BOOL;
		pusher_distance_5					:BOOL;
		pusher_distance_6					:BOOL;
		pusher_retract						:BOOL;
		
		compress_initial_speed				:BOOL;
		compress_initial_distance			:BOOL;
		compress_relax_distance				:BOOL;
		compress_retract_speed				:BOOL;
	END_STRUCT
END_TYPE

// ---- DUTs/Limits.TcDUT
TYPE Limits :
	STRUCT
		max_limit_Compress				:LREAL;
		max_limit_Shield				:LREAL;
		max_limit_Pusher 				:LREAL;
		max_pusher_shield_diff			:LREAL;
		max_torque						:LREAL;
	END_STRUCT
END_TYPE

// ---- DUTs/Rec_Compress.TcDUT
TYPE Rec_Compress :
	STRUCT
		Initial_Speed				:LREAL;
		Initial_Distance			:LREAL;
		Relax_Distance				:LREAL;
		Retract_Speed				:LREAL;
	END_STRUCT
END_TYPE

// ---- DUTs/Rec_Other.TcDUT
TYPE Rec_Other :
	STRUCT
		Compress_Home_Offset		:LREAL;
		Pusher_Home_Offset			:LREAL;
		Shield_Home_Offset			:LREAL;

	END_STRUCT
END_TYPE

// ---- DUTs/Rec_Pusher.TcDUT
TYPE Rec_Pusher :
	STRUCT
		//Initial_Speed				:LREAL;
		//Initial_Distance			:LREAL;
		//Eject_Speed					:LREAL;
		//Eject_Distance				:LREAL;
		//Retract_Speed				:LREAL;
		//tamp_initial_speed			:LREAL;
		//tamp_final_speed			:LREAL;
		//tamp_initial_distance		:LREAL;
		//tamp_final_distance			:LREAL;
		
		Speed				:ARRAY[1..6] OF LREAL;
		Distance			:ARRAY[1..6] OF LREAL;
		retract_speed			:LREAL;
		
	END_STRUCT
END_TYPE

// ---- DUTs/Rec_Clamp.TcDUT
TYPE Rec_Clamp :
	STRUCT
		Release_Instance				:LREAL;
	END_STRUCT
END_TYPE

// ---- DUTs/Rec_Shield.TcDUT
TYPE Rec_Shield :
	STRUCT
		//Initial_Speed			:LREAL;
		//Initial_Distance		:LREAL;
		//Retract_Speed			:LREAL;
		Speed					:ARRAY[1..6] OF LREAL;
		Distance				:ARRAY[1..6] OF LREAL;
		retract_speed			:LREAL;
		
	END_STRUCT
END_TYPE

// ---- DUTs/st_recipe_titles.TcDUT
TYPE st_recipe_titles :
	STRUCT
		pusher					:STRING;
		compress				:STRING;
		shield					:STRING;
		clamp					:STRING;
		offset					:STRING;
		
	END_STRUCT
END_TYPE

// ---- DUTs/st_yellow_visibility.TcDUT
TYPE st_yellow_visibility :
STRUCT
	main				:BOOL;
	recipe				:BOOL;
	graph				:BOOL;
	maintenance			:BOOL;
	io					:BOOL;
	auto_mode			:BOOL;
	debug_mode			:BOOL;
END_STRUCT
END_TYPE

// ---- GVLs/GVL_IO.TcGVL
VAR_GLOBAL
	CompressAxis :AXIS_REF;	
	PusherAxis :AXIS_REF;	
	ShieldAxis :AXIS_REF;	
	ResetLampController : FB_LampController;
	StartLampController : FB_LampController;
	
	Name_String	AT%IB10 :STRING;
	Name_DINT1	AT%IB10	:DINT;
		
	// Cabinet Digital Inputs 1 - Device 1, Term 2
	ixCabinetE_StopButtonOkay AT%IX0.0 :BOOL;
	ixE_StopRelayOkay AT%IX0.1 :BOOL;
	ixGuardRelayOkay AT%IX0.2 :BOOL;
	ixSpareIN4 AT%IX0.3 :BOOL;
	ixSpareIN5 AT%IX0.4 :BOOL;
	ixResetButton AT%IX0.5 :BOOL;
	ixSpareIN7 AT%IX0.6 :BOOL;
	ixSpareIN8 AT%IX0.7 :BOOL;
	ixStart_Button_Machine AT%IX1.0 :BOOL;
	ixStop_Button AT%IX1.1 :BOOL;
	ixSpareIN11 AT%IX1.2 :BOOL;
	ixSpareIN12 AT%IX1.3 :BOOL;
	ixSpareIN13 AT%IX1.4 :BOOL;
	ixSpareIN14 AT%IX1.5 :BOOL;
	ixSpareIN15 AT%IX1.6 :BOOL;
	ixSpareIN16 AT%IX1.7 :BOOL;
	
	// Cabinet Digital Outputs 1 - Device 1, Term 3
	qxEnableE_Stop AT%QX0.0 :BOOL;
	qxClamp		 AT%QX0.1 :BOOL :=FALSE;
	qxSpareOUT3 AT%QX0.2 :BOOL;
	qxStartButtonLamp AT%QX0.3:BOOL;
	qxResetButtonLamp AT%QX0.4 :BOOL;
	qxSpareOUT6 AT%QX0.5 :BOOL;
	qxSpareOUT7 AT%QX0.6 :BOOL;
	qxSpareOUT8 AT%QX0.7 :BOOL;
	
	// Servo Analogue Inputs 1- Device 2, Term 2
	ibCompressServoTorque AT%IB120 :INT;
	ibCompressServoFollowingError AT%IB124 :DINT;
	qbCompressServoTorqueLimit AT%QB120 :UINT;
	
	// Servo Analogue Inputs 1- Device 2, Term 3
	ibPusherServoTorque AT%IB130 :INT;
	ibPusherServoFollowingError AT%IB134 :DINT;
	qbPusherServoTorqueLimit AT%QB130 :UINT;
	
	// Servo Analogue Inputs 1- Device 2, Term 3
	ibShieldServoTorque AT%IB140 :INT;
	ibShieldServoFollowingError AT%IB144 :DINT;
	qbShieldServoTorqueLimit AT%QB140 :UINT;
	
	// Analogue Inputs - Device 2, Term 4
	(*iiAnalogueIn7_HeaterTemperature AT%IB112 :INT;
	iiAnalogueIn8_UserProbeTemperature AT%IB114 :INT;
	// Status Inputs - Device 2, Term 4
	ixHeaterTC_Error AT%IX2.0 :BOOL;
	ixUserTC_Error AT%IX2.1 :BOOL;*)
	
	// Machine Digital Inputs 1 - Device 2, Term 5
	ixCompressHomeSwitch AT%IX2.0 :BOOL;
	ixPusherHomeSwitch AT%IX2.1 :BOOL;
	ixShieldHomeSwitch AT%IX2.2 :BOOL;
	ixStartButton AT%IX2.3 :BOOL;
	ixSpareIN25 AT%IX2.4 :BOOL;
	ixspareIN26 AT%IX2.5 :BOOL;
	ixspareIN27 AT%IX2.6 :BOOL;
	ixSpareIN28 AT%IX2.7 :BOOL;
	ixGuardOkay AT%IX3.0 :BOOL;
	ixMachineE_StopButtonOkay AT%IX3.1 :BOOL;
	ixFanCartridgeDiagnostics AT%IX3.2 :BOOL;
	ixSpareIN32 AT%IX3.3 :BOOL;
	ixSpareIN33 AT%IX3.4 :BOOL;
	ixSpareIN34 AT%IX3.5 :BOOL;
	ixSpareIN35 AT%IX3.6 :BOOL;
	ixSpareIN36 AT%IX3.7 :BOOL;

	CompressServoErrorID: UDINT;
	PusherServoErrorID: UDINT;	
	ShieldServoErrorID: UDINT;
	
	sSystemStateHi : STRING;
	sSystemStateMed : STRING;
	sSystemStateLo : STRING;
	
END_VAR

// ---- GVLs/GVL_Objects.TcGVL
VAR_GLOBAL
	Clock 						: TClock;
	Config 						: TConfig;
	configuring					: BOOL;
	config_request				: BOOL;
	Config_Message				: STRING(300);
	config_speed				: INT:=1;
	List_of_Recipes				: ARRAY[1..10] OF Recipe;
END_VAR

// ---- GVLs/GVL_ZenOn.TcGVL
VAR_GLOBAL
	
	//graph visibility
	graph_visibility							:st_graph_visibility;
	yellow_visibility							:st_yellow_visibility;
	yellow_visibility_old						:st_yellow_visibility;

	overtorque_alarm							:BOOL;

	limits_screen								:Limits;
	limits_save									:Limits;
	save_limits									:BOOL:=FALSE;
	parameter_violation							:BOOL:=FALSE;

	//Mode
	Debug_Mode									:BOOL;
	
	//Recipe on the screen (current one)
	Recipe_Visibility							:ARRAY[1..10] OF BOOL:=[10(FALSE)];  //u are here
	

	
	Recipe_Screen								:Recipe;
	Default_Recipe_Visibility					:BOOL :=FALSE;
		
	//end_of_recipe_on_the_screen
	
	//Maintenance
	Maintenance_Visibility						:BOOL;
	Mode_String									:STRING;
	Stage_Name									:STRING;
	Step_Next									:BOOL;
	Toggle_Clamp								:BOOL;
	Force_Home									:BOOL;
	//end of maintenance
	
	//recipe functions
	SaveRecipe									:BOOL :=FALSE;
	SaveasRecipe								:BOOL :=FALSE;	
	
	
	
	LoadRecipe									:ARRAY[1..10] OF BOOL :=[10(FALSE)];
	Load_Request								:BOOL :=FALSE;
	Save_before_load							:BOOL :=FALSE;
	
	DeleteRecipe								:ARRAY[1..10] OF BOOL :=[10(FALSE)];
	Delete_Request								:BOOL :=FALSE;
	
	

	Saveas_name									:STRING;
	Message										:STRING(300);
	alarm_message								:STRING(300);	
	question									:STRING(300);
	//current_recipe_message						:STRING;
	recipe_titles								:st_recipe_titles;
	language									:st_language;
	
	
	//end of recipe functions
	
	sc_CompressServoErrorID: UDINT;
	sc_PusherServoErrorID: UDINT;
	sc_ShieldServoErrorID: UDINT;
	sc_sSystemStateHi: STRING;
	sc_sSystemStateMed: STRING;
	sc_sSystemStateLo: STRING;
	

	
	// Servo Analogue Inputs 1- Device 2, Term 2
	CompressServoTorque          	: INT;
	CompressServoFollowingError		: DINT;
	CompressServoTorqueLimit		: UINT;
	
	// Servo Analogue Inputs 1- Device 2, Term 3
	PusherServoTorque				: INT;
	PusherServoFollowingError		: DINT;
	PusherServoTorqueLimit			: UINT;
	
	// Servo Analogue Inputs 1- Device 2, Term 3
	ShieldServoTorque				: INT;
	ShieldServoFollowingError		: DINT;
	ShieldServoTorqueLimit			: UINT;
		

	
	(* Data For the Main Screen *)
	//CurrentProcessState				: STRING;			//Main Screen

	

	
	(* Data For the Settings Screen *)
	//CompressDisplay					: LREAL;		//Settings Screen
	//PusherDisplay					: LREAL;		//Settings Screen
	//ShieldDisplay					: LREAL;
	
	Zenon_Offset_Compress			:BOOL;
	Zenon_Offset_Shield				:BOOL;
	Zenon_Offset_Pusher				:BOOL;
				
	
	(* Digital IO *)
	CabinetE_StopButtonOkay			: BOOL;
	E_StopRelayOkay					: BOOL;
	GuardRelayOkay					: BOOL;
	ResetButton                     : BOOL;
	EnableE_Stop					: BOOL;
	StartButtonLamp					: BOOL;
	ResetButtonLamp					: BOOL;
	
	Clamp_Alarm						:BOOL;
	Clamp_Cooling					:BOOL;
	Clamp_State						:BOOL;
	
	CompressHomeSwitch  			:BOOL;
	PusherHomeSwitch 				:BOOL;
	ShieldHomeSwitch 				:BOOL;
	StartButton 					:BOOL;

	GuardOkay 						:BOOL;
	MachineE_StopButtonOkay 		:BOOL;
	FanCartridgeDiagnostics 		:BOOL;

	ResetLamp						: BOOL;			//Digital IO Screen
	
	LampTest						: BOOL;			//Digital IO Screen

	CompressAxisPosition			: LREAL;		//IO Screen
	PusherAxisPosition				: LREAL;
	ShieldAxisPosition				: LREAL;
	
	//main
	product_count					: INT:=0;
	auto_cycle_time					: LREAL;
	actual_cycle_rate				: LREAL;
	
	compress_settings				:st_compress_settings;

END_VAR

// ---- POUs/PRG_MAIN.TcPOU
PROGRAM PRG_MAIN
VAR

	//test: BOOL;
	//debug: INT;
	all_config_initialised: BOOL;
	FirstScan			  : BOOL:=TRUE;
	temp: INT;
	arda: INT;
	bruce: INT;
END_VAR

//Recipes
Clock();


		
IF Config.Initialised() AND bruce < 70 THEN
	bruce:=bruce+1;
ELSIF Config.Initialised() THEN   
	arda := arda+1;
	PRG_IO();
	PRG_Machine();
END_IF

FirstSCan:=FALSE;

END_PROGRAM

// ---- POUs/PRG_IO.TcPOU
PROGRAM PRG_IO
VAR
	
	//piccirix		:INT;
	TextTimer: ton;
	Message_timer: ton;
	actual_cycle_timer: ton;
	

	recipe_default				:recipe;
	Current_Recipe				:Recipe;
	empty_recipe				:Recipe;
	current_recipe_no			:INT:=1;
	saveas_recipe_no			:INT;
	load_recipe_no				:INT;
	delete_recipe_no			:INT;
	temp						:INT;
	temp2						:INT;
		
	Initialise					:BOOL := TRUE;
	InitialiseTickCounter		:INT;
	TickCounter					:INT;
	
	save_requested				:BOOL;
	
	Pusher_Home					:BOOL;
	Shield_Home					:BOOL;
	Compress_Home				:BOOL;
	
	//violation
	//old_recipe					:Recipe;
	//old_limits					:Limits;
	zero_violation				:BOOL;
	max_distance_violation		:BOOL;
	max_sh_push_diff_violation	:BOOL;
	
	Message_old					:STRING(300);
	
	Message_State				:INT:=0;
	
	//deleting					:BOOL;
	//saving						:BOOL;
	//saving_as					:BOOL;
	//saving_lim					:BOOL;
	
	done						:BOOL:=FALSE;
	//you are here!!!!!!!!!!
	
	//cycles_waited				:INT;
	product_count_old			:INT;
	actual_cycle_array			: ARRAY[1..10] OF LREAL;
	
	
END_VAR

VAR_OUTPUT
					
END_VAR

ResetLampController();
StartLampController();
Message_timer();
actual_cycle_timer();

done:=TRUE;
//old_recipe:=current_recipe;
f_initialisation();

f_param_violation();

f_calc_auto_cycle_time();

f_calc_actual_cycle_rate();

f_alarms();

f_save_as();

f_load();

f_delete();

f_save();

f_save_limits();

f_configure_recipe();

f_titles();

f_message_timer();

//end recipes
f_leftbar_visibility();

f_digital_io();
		
f_mode_of_operation();

METHOD f_alarms : BOOL
VAR_INPUT
END_VAR
IF zero_violation THEN
	IF language.english THEN
		alarm_message:='Some parameters can not be set to zero.'; 
	ELSE
		alarm_message:='Alguns parâmetros não podem ser ajustados para zero.';
	END_IF
END_IF

IF max_distance_violation THEN
	
	IF language.english THEN
		alarm_message:='Maximum axis distance violation';
	ELSE
		alarm_message:='Violação máxima da distância do eixo';
	END_IF 
END_IF

IF max_sh_push_diff_violation THEN
	
	
	IF language.english THEN
		alarm_message:='Maximum pusher-shield distance difference violation';
	ELSE
		alarm_message:='Violação máxima da diferença de distância entre proteção-empurrador';
	END_IF 
 
END_IF

IF Clamp_Alarm THEN
	
	
	IF language.english THEN
		alarm_message:='Clamp Overtime';
	ELSE
		alarm_message:='Tempo adicional de grampo';
	END_IF 
END_IF

IF Overtorque_alarm THEN
	
	
	IF language.english THEN
		alarm_message:='Motor Overtorque';
	ELSE
		alarm_message:='Excesso de torque do motor';
	END_IF
	
END_IF

IF NOT ixGuardOkay THEN
	
	
	IF language.english THEN
		alarm_message:='Guard Open';
	ELSE
		alarm_message:='Guarda Aberto';
	END_IF
END_IF

IF NOT CabinetE_StopButtonOkay THEN
	
	IF language.english THEN
		alarm_message:='E-Stop Pressed';
	ELSE
		alarm_message:='Parada de emergência pressionada';
	END_IF
END_IF

IF CabinetE_StopButtonOkay AND ixGuardOkay AND NOT parameter_violation AND NOT Overtorque_alarm AND NOT Clamp_Alarm THEN
	alarm_message:='';
END_IF
END_METHOD

METHOD f_calc_actual_cycle_rate : BOOL
VAR
	cropped_product_count			:INT;
	temp_for						:INT;
	total_time						:LREAL;
END_VAR
actual_cycle_timer.IN:=TRUE;
actual_cycle_timer.PT:= T#604800S; //week



IF actual_cycle_timer.Q THEN
	//cycles_waited:=cycles_waited+1;
	actual_cycle_timer.IN:=FALSE;


ELSIF product_count_old <> product_count THEN
	
	actual_cycle_array[10]:=actual_cycle_array[9];
	actual_cycle_array[9]:=actual_cycle_array[8];
	actual_cycle_array[8]:=actual_cycle_array[7];
	actual_cycle_array[7]:=actual_cycle_array[6];
	actual_cycle_array[6]:=actual_cycle_array[5];
	actual_cycle_array[5]:=actual_cycle_array[4];
	actual_cycle_array[4]:=actual_cycle_array[3];
	actual_cycle_array[3]:=actual_cycle_array[2];
	actual_cycle_array[2]:=actual_cycle_array[1];
	
	
	actual_cycle_array[1]:=(*cycles_waited*300+*)TIME_TO_LREAL(actual_cycle_timer.ET);
	//cycles_waited:=0;
	actual_cycle_timer.IN:=FALSE;
	
	
END_IF


cropped_product_count:=product_count;

IF cropped_product_count > 10 THEN
	cropped_product_count:=10;
END_IF 

IF cropped_product_count <>0 THEN
	
	total_time:=0;
	FOR temp_for := 1 TO cropped_product_count DO
		total_time:=total_time+actual_cycle_array[temp_for];
	END_FOR
	
	actual_cycle_rate := ((cropped_product_count*3600000)/total_time);
	
ELSE
	total_time:=0;
	actual_cycle_rate:=0;
END_IF



product_count_old:=product_count;
END_METHOD

METHOD f_calc_auto_cycle_time : BOOL
VAR
	shield_time			:LREAL;
	pusher_time			:LREAL;
	compress_time		:LREAL;
	temp				:LREAL;
	temp_pusher			:LREAL;
	temp_shield			:LREAL;

	
	temp_for			:INT;
	
	auto_time_array		:ARRAY [1..8] OF LREAL;
	
END_VAR

compress_time := recipe_screen.Compress.Initial_Distance/recipe_screen.compress.Initial_Speed;
temp:=ABS(recipe_screen.Compress.Initial_Distance-recipe_screen.Compress.Relax_Distance);
compress_time := compress_time + (temp/recipe_screen.compress.Initial_Speed);         
auto_time_array[1] := compress_time;

temp_shield:=0;
temp_pusher:=0;

FOR temp_for := 2 TO 7 DO

	shield_time:=(ABS(recipe_screen.Shield.Distance[temp_for-1]-temp_shield))/recipe_screen.Shield.Speed[temp_for-1];
	temp_shield:=recipe_screen.Shield.Distance[temp_for-1];
	
	pusher_time:=(ABS(recipe_screen.Pusher.Distance[temp_for-1]-temp_pusher))/recipe_screen.Pusher.Speed[temp_for-1];
	temp_pusher:=recipe_screen.Pusher.Distance[temp_for-1];
	
	IF pusher_time > shield_time THEN
		auto_time_array[temp_for]:=pusher_time;	
	ELSE
		auto_time_array[temp_for]:=shield_time;
	END_IF
	
END_FOR

compress_time := recipe_screen.Compress.Relax_Distance/recipe_screen.Compress.Retract_speed;
shield_time := recipe_screen.Shield.Distance[6]/recipe_screen.Shield.retract_speed;
pusher_time := recipe_screen.Pusher.distance[6]/recipe_screen.pusher.retract_speed;

IF compress_time>=shield_time AND compress_time>=pusher_time THEN
	auto_time_array[8]:=compress_time;
END_IF

IF pusher_time>=shield_time AND pusher_time>=compress_time THEN
	auto_time_array[8]:=pusher_time;
END_IF

IF shield_time>=pusher_time AND shield_time>=compress_time THEN
	auto_time_array[8]:=shield_time;
END_IF

auto_cycle_time:=0;
FOR temp_for := 1 TO 8 DO
	auto_cycle_time:= auto_time_array[temp_for]+auto_cycle_time;
	
END_FOR
END_METHOD

METHOD f_configure_recipe : BOOL
VAR_INPUT
END_VAR

FOR temp := 1 TO 11 DO
	IF save_requested = TRUE THEN
		Config.CopyGlobalRecipiesToConfig();
		config_request:=TRUE;
		save_requested:=FALSE;
	END_IF
END_FOR
END_METHOD

METHOD f_delete : BOOL
VAR_INPUT
END_VAR
FOR temp := 1 TO 10 DO
	IF DeleteRecipe[temp] = TRUE THEN
		delete_recipe_no := temp;
		DeleteRecipe[temp] := FALSE;
		
		IF language.english THEN
			question := CONCAT('Do you want to delete recipe ', List_of_Recipes[delete_recipe_no].Name);
			question := CONCAT(question,'?');
		ELSE
			question := CONCAT('Deseja excluir a receita ', List_of_Recipes[delete_recipe_no].Name);
			question := CONCAT(question,'?');
		END_IF
 
	END_IF
END_FOR

IF Delete_Request = TRUE THEN
	
	Delete_Request:=FALSE;
	
	configuring:=TRUE;
	
	current_recipe_no:=delete_recipe_no;
	
	IF language.english THEN
		Message := CONCAT('Deleting recipe ',List_of_Recipes[current_recipe_no].Name );
		Message := CONCAT(Message,'...');

		Config_Message := concat('Recipe ', List_of_Recipes[current_recipe_no].Name);
		Config_Message := concat(Config_Message,' has been deleted.');
	ELSE
		Message := CONCAT('Excluindo receita ',List_of_Recipes[current_recipe_no].Name );
		Message := CONCAT(Message,'...');

		Config_Message := concat('A receita ', List_of_Recipes[current_recipe_no].Name);
		Config_Message := concat(Config_Message,' foi excluída.');
	END_IF
	
	WHILE (delete_recipe_no<10) AND List_of_Recipes[delete_recipe_no+1].Memory_Free = FALSE DO
		List_of_Recipes[delete_recipe_no]:=List_of_Recipes[delete_recipe_no+1];
		//save_requested[delete_recipe_no] := TRUE;
		delete_recipe_no:=delete_recipe_no+1;
	END_WHILE
	
	List_of_Recipes[delete_recipe_no] := empty_recipe;
	save_requested := TRUE;
	//List_of_Recipes[delete_recipe_no].Memory_Free:=FALSE;
	
	
	IF current_recipe_no = delete_recipe_no AND current_recipe_no <> 1 THEN
		current_recipe_no := current_recipe_no - 1;
	END_IF
		
	Current_Recipe := List_of_Recipes[current_recipe_no];
	recipe_screen:=current_recipe;
	
	
	
END_IF
END_METHOD

METHOD f_digital_io : BOOL
VAR_INPUT
END_VAR

(***************************** Data For the Main Screen ***********************)


CabinetE_StopButtonOkay := ixCabinetE_StopButtonOkay;
E_StopRelayOkay:=ixE_StopRelayOkay;
GuardRelayOkay:=ixGuardRelayOkay;
GuardOkay:=ixGuardOkay;

ResetButton := ixResetButton;

		
// Cabinet Digital Outputs 1 - Device 1, Term 3
EnableE_Stop:=qxEnableE_Stop;
	
//StartButtonLamp:=qxStartButtonLamp;
ResetButtonLamp:=qxResetButtonLamp;
	
	
// Servo Analogue Inputs 1- Device 2, Term 2
CompressServoTorque:=ibCompressServoTorque;
CompressServoFollowingError:=ibCompressServoFollowingError;
CompressServoTorqueLimit:=qbCompressServoTorqueLimit;
	
// Servo Analogue Inputs 1- Device 2, Term 3
PusherServoTorque:=ibPusherServoTorque;
PusherServoFollowingError:=ibPusherServoFollowingError;
PusherServoTorqueLimit:=qbPusherServoTorqueLimit;
	
// Servo Analogue Inputs 1- Device 2, Term 3
ShieldServoTorque:=ibShieldServoTorque;
ShieldServoFollowingError:=ibShieldServoFollowingError;
ShieldServoTorqueLimit:=qbShieldServoTorqueLimit;
	

	
// Machine Digital Inputs 1 - Device 2, Term 5
CompressHomeSwitch:=ixCompressHomeSwitch;
PusherHomeSwitch:=ixPusherHomeSwitch;
ShieldHomeSwitch:=ixShieldHomeSwitch;
StartButton:= ixStartButton;
GuardOkay:=ixGuardOkay; 
MachineE_StopButtonOkay:=ixMachineE_StopButtonOkay;
//FanCartridgeDiagnostics:=ixFanCartridgeDiagnostics;

//sc_CompressServoErrorID := CompressServoErrorID;
//sc_PusherServoErrorID := PusherServoErrorID;	
//sc_ShieldServoErrorID := ShieldServoErrorID;
	

//Homed?
Pusher_Home:=PRG_Machine.Pusher.HomeExecuted;
Shield_Home:=PRG_Machine.Shield.HomeExecuted;
Compress_Home:=PRG_Machine.Compress.HomeExecuted;
	
//Clamp
Clamp_State:=qxClamp;


qxResetButtonLamp := ResetLampController.Q; //io
ResetLamp := ResetLampController.Q; //zenon



ShieldAxisPosition := PRG_Machine.Shield.ShieldServo.fActualPosition;		
PusherAxisPosition := PRG_Machine.Pusher.PusherServo.fActualPosition;
CompressAxisPosition := PRG_Machine.Compress.CompressServo.fActualPosition;

Zenon_Offset_Compress:=PRG_Machine.Compress.OffsetExecuted;
Zenon_Offset_Shield:=PRG_Machine.Shield.OffsetExecuted;
Zenon_Offset_Pusher:=PRG_Machine.Pusher.OffsetExecuted;
END_METHOD

METHOD f_initialisation : BOOL
VAR
	//temp			:INT;
	
END_VAR

IF Initialise THEN
	//InitialiseTickCounter := InitialiseTickCounter + 1;
	//IF InitialiseTickCounter = 150 THEN
	//	Config.CopyConfigRecipiesToGlobal();
	//END_IF
	//piccirix:=piccirix+1;
	
	Config.CopyConfigRecipiesToGlobal();
		//piccirix:=piccirix+1;
	
	//piccirix:=piccirix+1;	
	//IF InitialiseTickCounter >= 300 THEN	
	//recipe_screen := List_of_Recipes[1];
	yellow_visibility.main:=TRUE;
	
	recipe_default.Name:='default 1';
	
	recipe_default.Compress.Initial_Distance:=5;
	recipe_default.Compress.Initial_Speed:=5;
	recipe_default.Compress.Relax_Distance:=3;
	recipe_default.Compress.Retract_Speed:=5;
	
	recipe_default.Pusher.Speed[1]:=5;
	recipe_default.Pusher.Speed[2]:=5;
	recipe_default.Pusher.Speed[3]:=5;
	recipe_default.Pusher.Speed[4]:=5;
	recipe_default.Pusher.Speed[5]:=5;
	recipe_default.Pusher.Speed[6]:=5;
	recipe_default.Pusher.Retract_Speed:=5;
	recipe_default.Pusher.Distance[1]:=5;
	recipe_default.Pusher.Distance[2]:=0;
	recipe_default.Pusher.Distance[3]:=5;
	recipe_default.Pusher.Distance[4]:=0;
	recipe_default.Pusher.Distance[5]:=5;
	recipe_default.Pusher.Distance[6]:=0;

	recipe_default.Shield.Speed[1]:=5;
	recipe_default.Shield.Speed[2]:=5;
	recipe_default.Shield.Speed[3]:=5;
	recipe_default.Shield.Speed[4]:=5;
	recipe_default.Shield.Speed[5]:=5;
	recipe_default.Shield.Speed[6]:=5;
	recipe_default.Shield.Retract_Speed:=5;
	recipe_default.Shield.Distance[1]:=5;
	recipe_default.Shield.Distance[2]:=0;
	recipe_default.Shield.Distance[3]:=5;
	recipe_default.Shield.Distance[4]:=0;
	recipe_default.Shield.Distance[5]:=5;
	recipe_default.Shield.Distance[6]:=0;
	
	recipe_default.Other.Compress_Home_Offset:=3;
	recipe_default.Other.Pusher_Home_Offset:=3;
	recipe_default.Other.Shield_Home_Offset:=3;
	
	recipe_default.Memory_Free:=FALSE;
	
	List_of_Recipes[1]:=recipe_default;
	recipe_screen:=List_of_Recipes[1];	
		
	limits_screen:=limits_save;
	
	IF language.english THEN
		Message:='Welcome!';
	ELSE
		Message:='Bem-vindo!';
	END_IF
	
	InitialiseTickCounter := 0;
	Initialise := FALSE;
	//END_IF		
ELSE
	//InitialiseTickCounter := 0;
	
	//FOR temp:=1 TO 11 DO
	///	Config.CopyConfigRecipiesToGlobal(temp);
		//piccirix:=piccirix+1;
	//END_FOR

	current_recipe:=recipe_screen;

	//current_recipe_message:=CONCAT('The current recipe number is ',INT_TO_STRING(Current_recipe_no));
	
	IF current_recipe_no = 1 THEN
		Default_Recipe_Visibility:=FALSE;
	ELSE
		Default_Recipe_Visibility:=TRUE;
	END_IF
	
	FOR	temp := 1 TO 10 DO
		Recipe_Visibility[temp]:=NOT(List_of_Recipes[temp].Memory_Free);
	END_FOR
	
	//temp:=1;
END_IF
END_METHOD

METHOD f_leftbar_visibility : BOOL
VAR_INPUT
END_VAR
IF NOT yellow_visibility_old.main AND yellow_visibility.main THEN
	yellow_visibility.recipe:=FALSE;
	yellow_visibility.maintenance:=FALSE;
	yellow_visibility.io:=FALSE;
	yellow_visibility.graph:=FALSE;
		
END_IF

IF NOT yellow_visibility_old.recipe AND yellow_visibility.recipe THEN
	yellow_visibility.main:=FALSE;
	yellow_visibility.maintenance:=FALSE;
	yellow_visibility.io:=FALSE;
	yellow_visibility.graph:=FALSE;
		
END_IF

IF NOT yellow_visibility_old.graph AND yellow_visibility.graph THEN
	yellow_visibility.main:=FALSE;
	yellow_visibility.maintenance:=FALSE;
	yellow_visibility.io:=FALSE;
	yellow_visibility.recipe:=FALSE;
		
END_IF

IF NOT yellow_visibility_old.io AND yellow_visibility.io THEN
	yellow_visibility.main:=FALSE;
	yellow_visibility.maintenance:=FALSE;
	yellow_visibility.graph:=FALSE;
	yellow_visibility.recipe:=FALSE;
		
END_IF

IF NOT yellow_visibility_old.maintenance AND yellow_visibility.maintenance THEN
	yellow_visibility.main:=FALSE;
	yellow_visibility.io:=FALSE;
	yellow_visibility.graph:=FALSE;
	yellow_visibility.recipe:=FALSE;
		
END_IF

yellow_visibility_old.main:=yellow_visibility.main;
yellow_visibility_old.maintenance:=yellow_visibility.maintenance;
yellow_visibility_old.recipe:=yellow_visibility.recipe;
yellow_visibility_old.graph:=yellow_visibility.graph;
yellow_visibility_old.io:=yellow_visibility.io;
END_METHOD

METHOD f_load : BOOL
VAR_INPUT
END_VAR
FOR temp := 1 TO 10 DO
	IF LoadRecipe[temp] = TRUE THEN
		load_recipe_no := temp;
		LoadRecipe[temp] := FALSE;
		

		
		IF language.english THEN
			question := CONCAT('Do you want to save recipe ', recipe_screen.Name);
			question := CONCAT(question,', before loading the recipe ');
			question := CONCAT(question, List_of_Recipes[load_recipe_no].Name);
			question := CONCAT(question,'?');			
		ELSE
			question := CONCAT('Deseja salvar a receita ', recipe_screen.Name);
			question := CONCAT(question,', antes de carregar a receita ');
			question := CONCAT(question, List_of_Recipes[load_recipe_no].Name);
			question := CONCAT(question,'?');			
		END_IF
 		
	END_IF
END_FOR

IF Load_Request = TRUE THEN
	
	Load_Request:=FALSE;
	
	IF(Save_before_load=TRUE)THEN
		
		configuring:=TRUE;
		//current_recipe:=recipe_screen;
		List_of_Recipes[current_recipe_no] := current_recipe;
		List_of_Recipes[current_recipe_no].Memory_Free := FALSE;
		//config.CopySettingsFromGlobal();
		Save_before_load := FALSE;
		
		IF language.english THEN
			Message := CONCAT('Saving recipe ',recipe_screen.Name);
			Message := CONCAT(Message,'... ');
		
			Config_Message := concat('Recipe ', recipe_screen.Name);
			Config_Message := concat(Config_Message,' has been saved.');
		ELSE
			
			Message := CONCAT('Salvando receita ',recipe_screen.Name);
			Message := CONCAT(Message,'... ');
		
			Config_Message := concat('A receita ', recipe_screen.Name);
			Config_Message := concat(Config_Message,' foi salva.');			
		END_IF
		save_requested := TRUE;	
		
	ELSE
		IF language.english THEN
			Message := CONCAT('Recipe ',List_of_Recipes[load_recipe_no].Name);
			Message := CONCAT(Message,' has been loaded');
		ELSE
			Message := CONCAT('A receita ',List_of_Recipes[load_recipe_no].Name);
			Message := CONCAT(Message,' foi carregada.');			
		END_IF
	END_IF
	
	current_recipe_no:=load_recipe_no;
		
	Current_Recipe := List_of_Recipes[current_recipe_no];
	recipe_screen:=current_recipe;
	//Message := CONCAT('Recipe ',current_recipe.Name);
	//Message := CONCAT(Message,' loading... ');

	
END_IF
END_METHOD

METHOD f_message_timer : BOOL
VAR_INPUT
END_VAR
CASE Message_State OF

0:
	
	IF Message <> message_old THEN
		//Message_State:=2;
		Message_timer.IN:=FALSE;
		Message_Timer.PT:=T#10S;
		Message_State:=0;
		
		Message_State:=1;
		
	END_IF
1:
	Message_timer.IN:=TRUE;
	Message_Timer.PT:=T#10S;
	Message_State:=0;
END_CASE

IF Message_Timer.Q = TRUE THEN
	Message:='';
	Message_timer.IN:=FALSE;
	Message_Timer.PT:=T#10S;
	//Message_Timer.PT:=T#30S;
END_IF 
Message_old:=Message;
END_METHOD

METHOD f_mode_of_operation : BOOL
VAR_INPUT
END_VAR
//Mode
IF debug_mode = FALSE THEN
	IF language.english THEN
		mode_string:= 'Current Mode: Automatic';
	ELSE
		mode_string:= 'Modo atual: Automático';
	END_IF
	yellow_visibility.auto_mode:=TRUE;
	yellow_visibility.debug_mode:=FALSE;
ELSE
	IF language.english THEN
		mode_string:= 'Current Mode: Debug';
	ELSE
		mode_string:= 'Modo atual: Depuração';
	END_IF
	yellow_visibility.auto_mode:=FALSE;
	yellow_visibility.debug_mode:=TRUE;
END_IF

//until here
END_METHOD

METHOD f_param_violation : BOOL
VAR
	pusher_calc				:ARRAY[0..6] OF LREAL;
	shield_calc				:ARRAY[0..6] OF LREAL;
	pusher_time				:LREAL;
	shield_time				:LREAL;
END_VAR
//violation

IF  
	recipe_screen.Compress.Initial_Speed =0 OR 
	recipe_screen.Compress.Retract_Speed =0 OR
	recipe_screen.pusher.speed[1] = 0 OR
	recipe_screen.pusher.speed[2] = 0 OR
	recipe_screen.pusher.speed[3] = 0 OR
	recipe_screen.pusher.speed[4] = 0 OR
	recipe_screen.pusher.speed[5] = 0 OR
	recipe_screen.pusher.speed[6] = 0 OR
	recipe_screen.Pusher.Retract_Speed = 0 OR
	recipe_screen.Shield.speed[1] = 0 OR
	recipe_screen.Shield.speed[2] = 0 OR
	recipe_screen.Shield.speed[3] = 0 OR
	recipe_screen.Shield.speed[4] = 0 OR
	recipe_screen.Shield.speed[5] = 0 OR
	recipe_screen.Shield.speed[6] = 0 OR
	recipe_screen.Shield.Retract_Speed = 0 THEN
		
	zero_violation := TRUE;
		
ELSE
	zero_violation := FALSE;
END_IF

IF 	recipe_screen.Other.Compress_Home_Offset > limits_screen.max_limit_compress OR
	recipe_screen.Other.Shield_Home_Offset > limits_screen.max_limit_Shield OR
	recipe_screen.Other.Pusher_Home_Offset > limits_screen.max_limit_Pusher OR
	
	recipe_screen.Compress.Initial_Distance + recipe_screen.Other.Compress_Home_Offset > limits_screen.max_limit_compress OR
	recipe_screen.Compress.Relax_Distance + recipe_screen.Other.Compress_Home_Offset > limits_screen.max_limit_compress OR
	
	recipe_screen.Shield.Distance[1] + recipe_screen.Other.shield_Home_Offset > limits_screen.max_limit_shield OR
	recipe_screen.Shield.Distance[2] + recipe_screen.Other.shield_Home_Offset > limits_screen.max_limit_shield OR
	recipe_screen.Shield.Distance[3] + recipe_screen.Other.shield_Home_Offset > limits_screen.max_limit_shield OR
	recipe_screen.Shield.Distance[4] + recipe_screen.Other.shield_Home_Offset > limits_screen.max_limit_shield OR
	recipe_screen.Shield.Distance[5] + recipe_screen.Other.shield_Home_Offset > limits_screen.max_limit_shield OR
	recipe_screen.Shield.Distance[6] + recipe_screen.Other.shield_Home_Offset > limits_screen.max_limit_shield OR
	
	recipe_screen.Pusher.Distance[1] + recipe_screen.Other.Pusher_Home_Offset > limits_screen.max_limit_pusher OR
	recipe_screen.Pusher.Distance[2] + recipe_screen.Other.Pusher_Home_Offset > limits_screen.max_limit_pusher OR
	recipe_screen.Pusher.Distance[3] + recipe_screen.Other.Pusher_Home_Offset > limits_screen.max_limit_pusher OR
	recipe_screen.Pusher.Distance[4] + recipe_screen.Other.Pusher_Home_Offset > limits_screen.max_limit_pusher OR
	recipe_screen.Pusher.Distance[5] + recipe_screen.Other.Pusher_Home_Offset > limits_screen.max_limit_pusher OR
	recipe_screen.Pusher.Distance[6] + recipe_screen.Other.Pusher_Home_Offset > limits_screen.max_limit_pusher THEN
	
	max_distance_violation:=TRUE;
	
ELSE
	max_distance_violation:=FALSE;
END_IF

max_sh_push_diff_violation := FALSE;

pusher_calc[0]:=recipe_screen.Other.Pusher_Home_Offset;
shield_calc[0]:=recipe_screen.Other.shield_Home_Offset;

FOR temp:=1 TO 6 DO
	pusher_calc[temp]:=recipe_screen.Other.Pusher_Home_Offset + recipe_screen.Pusher.Distance[temp];
	shield_calc[temp]:=recipe_screen.Other.Shield_Home_Offset + recipe_screen.Shield.Distance[temp];
END_FOR


FOR temp:=0 TO 6 DO
	IF pusher_calc[temp]-shield_calc[temp]> limits_screen.max_pusher_shield_diff THEN
		max_sh_push_diff_violation := TRUE;
	END_IF                         
END_FOR

FOR temp:=0 TO 5 DO
	pusher_time:=(pusher_calc[temp+1]-pusher_calc[temp])/recipe_screen.Pusher.Speed[temp+1];
	shield_time:=(shield_calc[temp+1]-shield_calc[temp])/recipe_screen.Shield.Speed[temp+1];
	IF recipe_screen.Pusher.Speed[temp+1] > recipe_screen.Shield.Speed[temp+1] AND pusher_time < shield_time THEN
    	IF pusher_calc[temp+1]-(pusher_time*recipe_screen.Shield.Speed[temp+1]+shield_calc[temp]) > limits_screen.max_pusher_shield_diff  THEN
			max_sh_push_diff_violation := TRUE;
		END_IF	
	
			
	END_IF                         
END_FOR


IF max_sh_push_diff_violation OR max_distance_violation OR zero_violation THEN
	parameter_violation:=TRUE;
ELSE
	parameter_violation:=FALSE;
END_IF


//violation end
END_METHOD

METHOD f_save : BOOL
VAR_INPUT
END_VAR
IF SaveRecipe THEN
	SaveRecipe := FALSE;

	current_recipe.Memory_Free:=FALSE;
	configuring:=TRUE;
	
	IF language.english THEN
		Message :=concat('Saving Recipe ',current_recipe.Name);	
		Message :=concat(Message,'...');
	
		Config_Message := concat('Recipe ', current_recipe.Name);
		Config_Message := concat(Config_Message,' has been saved.');
	ELSE
		Message :=concat('Salvando receita ',current_recipe.Name);	
		Message :=concat(Message,'...');
	
		Config_Message := concat('A receita ', current_recipe.Name);
		Config_Message := concat(Config_Message,' foi salva');
	END_IF
	
	List_of_Recipes[current_recipe_no] := current_recipe;
	save_requested := TRUE;
	
END_IF
END_METHOD

METHOD f_save_as : BOOL
VAR_INPUT
END_VAR
IF SaveasRecipe = TRUE THEN
	saveas_recipe_no:=current_recipe_no;
	WHILE (List_of_Recipes[saveas_recipe_no].Memory_Free = FALSE) AND (saveas_recipe_no<11) DO  
		saveas_recipe_no:=saveas_recipe_no+1;
		
	END_WHILE
	
	IF saveas_recipe_no > 10 THEN
		
		IF language.english THEN
			Message:='Maximum Recipe limit has been reached.';
		ELSE
			Message:='A limite máxima de receita foi alcançada.';
		END_IF
		
		saveas_recipe_no:=10;
		SaveasRecipe := FALSE;	
	
		
	ELSIF List_of_Recipes[saveas_recipe_no].Memory_Free = TRUE THEN
		SaveasRecipe:=FALSE;
		
		IF language.english THEN
			Message :=concat( 'Recipe ',current_recipe.Name);
			Message :=concat( Message,' is being saved as ');
			Message :=concat( Message,saveas_name);
			Message :=concat( Message,'...');
		
			Config_Message := concat('Recipe ', current_recipe.Name);
			Config_Message := concat(Config_Message,' has been saved as ');
			Config_Message := concat(Config_Message,saveas_name);
			Config_Message := concat(Config_Message,'.');
		ELSE //ure here........
			Message :=concat( 'A receita ',current_recipe.Name);
			Message :=concat( Message,' está sendo salva como ');
			Message :=concat( Message,saveas_name);
			Message :=concat( Message,'...');
		
			Config_Message := concat('A receita ', current_recipe.Name);
			Config_Message := concat(Config_Message,' foi salva como receita ');
			Config_Message := concat(Config_Message,saveas_name);
			Config_Message := concat(Config_Message,'.');			
		END_IF
		
		configuring:=TRUE;
		save_requested := TRUE;

		List_of_Recipes[saveas_recipe_no]:=current_recipe;
		List_of_Recipes[saveas_recipe_no].Name:=Saveas_name;
		List_of_Recipes[saveas_recipe_no].Memory_Free:=FALSE;
		//current_recipe:=recipe_screen;
		//Config.CopyGlobalRecipiesToConfig();
		
		//Current_Recipe := List_of_Recipes[current_recipe_no];
		//recipe_screen:=current_recipe;

				
	
	END_IF
	
END_IF
END_METHOD

METHOD f_save_limits : BOOL
VAR_INPUT
END_VAR
IF save_limits THEN
	save_limits:=FALSE;
	limits_save:=limits_screen;
	save_requested := TRUE;
	
	IF language.english THEN
		Message:='Saving Limits...';
	ELSE
		Message:='Salvando limites...';
	END_IF
		
	Config_Message:='Limits has been saved';
	configuring:=TRUE;
END_IF
END_METHOD

METHOD f_titles : BOOL
VAR_INPUT
END_VAR

IF language.english THEN
	recipe_titles.clamp:=concat( 'Clamp parameters for recipe ',recipe_screen.Name); 
	recipe_titles.clamp:=concat( recipe_titles.clamp,':');
ELSE
	recipe_titles.clamp:=concat( 'Parâmetros do grampo para receita ',recipe_screen.Name); 
	recipe_titles.clamp:=concat( recipe_titles.clamp,':');
END_IF

IF language.english THEN
	recipe_titles.compress:=concat( 'Compress parameters for recipe ',recipe_screen.Name); 
	recipe_titles.compress:=concat( recipe_titles.compress,':');
ELSE
	recipe_titles.compress:=concat( 'Parâmetros de compressão para receita ',recipe_screen.Name); 
	recipe_titles.compress:=concat( recipe_titles.compress,':');	
END_IF

IF language.english THEN
	recipe_titles.offset:=concat( 'Offset parameters for recipe receita ',recipe_screen.Name); 
	recipe_titles.offset:=concat( recipe_titles.offset,':');
ELSE
	recipe_titles.offset:=concat( 'Parâmetros de desvio para receita ',recipe_screen.Name); 
	recipe_titles.offset:=concat( recipe_titles.offset,':');
END_IF

IF language.english THEN
	recipe_titles.shield:=concat( 'Shield parameters for recipe ',recipe_screen.Name); 
	recipe_titles.shield:=concat( recipe_titles.shield,':');
ELSE
	recipe_titles.shield:=concat( 'Parâmetros de proteção para receita ',recipe_screen.Name); 
	recipe_titles.shield:=concat( recipe_titles.shield,':');
END_IF

IF language.english THEN
	recipe_titles.pusher:=concat( 'Pusher parameters for recipe ',recipe_screen.Name); 
	recipe_titles.pusher:=concat( recipe_titles.pusher,':');
ELSE
	recipe_titles.pusher:=concat( 'Parâmetros do empurrador para receita ',recipe_screen.Name); 
	recipe_titles.pusher:=concat( recipe_titles.pusher,':');
END_IF
END_METHOD

END_PROGRAM

// ---- POUs/PRG_Machine.TcPOU
PROGRAM PRG_Machine
VAR
	
	//empty recipe
	empty_recipe				:recipe;
	
	//debug
	after_debug_state					:INT :=0;

	
	Pusher :FB_Pusher;
	Compress: FB_Compress;
	Shield: FB_Shield;

	ZenonStart: NT_StartProcess;

	
	debug_counter: INT;
	tickcounter: INT;
	tickcounter2: INT;

	State: INT:= 0;
	state_old: INT:=0;
	StateNext: INT:= 0;
	
	SM_StepRequest: BOOL:=FALSE;
	singleStep: BOOL:=FALSE;
		
	Clamp_Security_Time: TIME := T#30S;
	ClampTimer: TON;
	//DwellTimer: TON;
	//SaveTickCounter: INT := 0;

	DatumTaught: BOOL;

	

	
	//stage
	stage_sh_push						:INT:=1;
	
END_VAR

VAR_OUTPUT

	rec_old		:recipe;
END_VAR

IF TRUE THEN
	debug_counter := debug_counter+1;
END_IF



qbCompressServoTorqueLimit := 1000;
qbPusherServoTorqueLimit := 1000;
qbShieldServoTorqueLimit := 1000;


//The state-machine
CASE State OF
	
0: //Copy config .txt file into machine settings
	


	//Zenon start process function call - appears to never generate errors
	
	//IF ZenonStart.Busy=FALSE THEN
	ZenonStart (
		NETID :=,
		//PATHSTR := 'Hard Disk\CP6606_Runtime\zenonRCE.exe', //'C:\PROGRAM Files\COPA-DATA\zenon 7.20 SP0\Zenrt32.exe',
		//DIRNAME := 'Hard Disk\CP6606_Runtime',  //'C:\Program Files\COPA-DATA\zenon 7.20 SP0',
		PATHSTR := 'Hard Disk\ZenonRunTime\zenonRCE.exe', //'C:\PROGRAM Files\COPA-DATA\zenon 7.20 SP0\Zenrt32.exe',
		DIRNAME := 'Hard Disk\ZenonRunTime',  //'C:\Program Files\COPA-DATA\zenon 7.20 SP0',
		COMNDLINE := '',
		START := TRUE,
		TMOUT := DEFAULT_ADS_TIMEOUT
		);
	StateNext := 10;



10: 
	qxEnableE_Stop := FALSE;
	tickcounter := 0;
	StateNext := 15;

15: //Check E-Stop relay is not set then Enable and initialise stuff - disable drive to clear errors

	

	//IF ixCabinetE_StopButtonOkay THEN
	qxEnableE_Stop := TRUE;
	StateNext := 20;
	//ELSE
	//	ResetLampController.State := SlowFlash;
	//END_IF
	
20: // Look for E-Stop button reset
	IF ixCabinetE_StopButtonOkay THEN
		//ResetLampController.State := steady;
		StateNext := 30;
	ELSE
		 
		ResetLampController.State := SlowFlash;
			
	END_IF
	
	//here
30: // Wait for operator to hit reset button
	
	IF ixE_StopRelayOkay THEN
		ResetLampController.State := off;
		StateNext := 40;
		tickcounter := 0;
	ELSE
		ResetLampController.State := steady;
		


	END_IF

40: // look for guard closed - disable drive to clear errors
	//sSystemStateMed := F_DisplayText("Guard Open",0);	
	//CurrentProcessState	:= F_DisplayText("not ready",0);	//Main Screen	

	
	IF NOT ixGuardOkay THEN
		ResetLampController.State := FastFlash;		
	ELSE
		ResetLampController.State := off;
		//sSystemStateMed := F_DisplayText("Initialising Axes",0);	
		tickcounter := 0;
		StateNext := 50;
	END_IF

50:
	IF ixGuardRelayOkay THEN
		statenext:=100;
	END_IF
	
100: // wait 2 scans for power supply to drive to stabilise
	tickcounter := tickcounter + 1;
	IF tickcounter >= 2 THEN
		tickcounter := 0;
		StateNext := 105;
	END_IF

105:
	IF NOT ixresetbutton THEN
		statenext:=110;
	END_IF	
	
110: // prepare for Servo motion - enable drive
//you are here!!!!!!!!!!!!!!!!!!!!!!!!!!!!
	//IF NOT ixResetButton THEN
		
		
	
	Shield._Enable();
	Pusher._Enable();
	Compress._Enable();
		
	tickcounter := tickcounter + 1;
	IF tickcounter >= 100 THEN
		tickcounter := 0;

		StateNext := 115;
	END_IF	
	//END_IF


	
115: 
	
	//IF Shield.HomeExecuted = FALSE OR Pusher.HomeExecuted = FALSE OR Compress.HomeExecuted = FALSE THEN
	IF language.english THEN
		Stage_Name := 'Beginning';
	ELSE
		Stage_Name := 'Início';
	END_IF
	Maintenance_Visibility:=TRUE;
	qxStartButtonLamp:=TRUE;
	IF (ixStartButton OR Step_Next OR ixStart_Button_Machine) THEN
		IF (parameter_violation = FALSE) THEN
			qxStartButtonLamp:=FALSE;
			StateNext := 116;
			Step_Next := FALSE;
			Clamp_Alarm:=FALSE;
			Maintenance_Visibility:=FALSE;
			stage_sh_push:=1;
			//Stage_Name := 'Homing and Offsetting';



		ELSE
			Step_Next:=FALSE;
		END_IF
	END_IF

	
116:
	IF (NOT ixstartbutton) AND NOT ixstart_button_machine THEN
		//general_offset_update();

		
		statenext:=117;
	END_IF
	
117:
	IF Compress.HomeExecuted=TRUE AND 
	   Shield.HomeExecuted = TRUE AND 
	   Pusher.HomeExecuted = TRUE AND
	   Pusher.OffsetExecuted = TRUE AND
	   Shield.OffsetExecuted = TRUE AND
	   Compress.OffsetExecuted = TRUE AND
	   Debug_Mode = FALSE THEN
	   
	   statenext:= 130;
	ELSE
		statenext:=120;
	END_IF
	
	Shield.Shield_param:=recipe_screen;
	Compress.Compress_Param := recipe_screen;
	Pusher.Pusher_Param := recipe_screen;
	//ELSE
	//	StateNext:=129;
	//	after_debug_state:=128;
	//END_IF
		
120: //you are here!!!!!!!!!!!!

	IF language.english THEN
		Stage_Name := 'Homing';
	ELSE
		Stage_Name := 'Ir para Início';
	END_IF
	IF Pusher.HomeExecuted = FALSE THEN 
		Pusher._Home();
	END_IF
	
	IF Compress.HomeExecuted = FALSE THEN
		Compress._Home();
	END_IF
	
	
	IF Compress.HomeExecuted AND Pusher.HomeExecuted THEN
		StateNext := 125;                //directly to end
		//Compress.HomeExecuted:=FALSE;
		//Pusher.HomeExecuted:=FALSE;
		
	END_IF
	
125:
	//random:='arda';
	IF Shield.HomeExecuted = FALSE THEN
		Shield._Home();
		
	ELSE
		StateNext := 129;
		IF language.english THEN
			Stage_Name := 'Homing done';
		ELSE
			Stage_Name := 'Ir para início concluído';
		END_IF
		after_debug_state :=127;
		//Shield.HomeExecuted := FALSE;
	END_IF

127:
	
	IF language.english THEN	
		Stage_Name := 'Offsetting';
	ELSE
		Stage_Name := 'Desviando';
	END_IF
	
	IF Compress.OffsetExecuted = FALSE THEN
		Compress.Offset(enable:=TRUE);
	END_IF
	
	IF Shield.OffsetExecuted = FALSE THEN
		Shield.Offset(enable:=TRUE);
	END_IF
	
	IF Pusher.OffsetExecuted = FALSE THEN
		Pusher.Offset(enable:=TRUE);
	END_IF
	
	IF Pusher.OffsetExecuted AND Shield.OffsetExecuted AND Compress.OffsetExecuted THEN
		Pusher.Offset(enable:=FALSE);
		Shield.Offset(enable:=FALSE);
		Compress.Offset(enable:=FALSE);
		
		rec_old:=Shield.Shield_Param;     //old values
		
		IF language.english THEN
			Stage_Name := 'Offsetting done';
		ELSE
			Stage_Name :='Desvio concluído';	
		END_IF
		
		Maintenance_Visibility := TRUE;
		qxStartButtonLamp:=TRUE;
		IF (ixStartButton OR Step_Next OR ixStart_Button_Machine) THEN
			IF (parameter_violation =FALSE) THEN
				qxStartButtonLamp:=FALSE;
				
				Shield.Shield_param:=recipe_screen;
				Compress.Compress_Param := recipe_screen;
				Pusher.Pusher_Param := recipe_screen;
			
				StateNext:=128;
				Step_Next:=FALSE;
				Maintenance_Visibility := FALSE;
			ELSE
				Step_Next:=FALSE;
			END_IF
		END_IF
	END_IF
	
128:	
	IF NOT ixstartbutton AND NOT ixstart_button_machine THEN
		statenext:=130;
	END_IF	

129: //debug	
	
	IF _debug(enable:=TRUE) THEN
		_debug(enable:=FALSE);
		statenext:=131;
	END_IF
		
130: //stage 1

	//IF ixstartbutton AND NOT ixstart_button_machine THEN
	IF language.english THEN
		Stage_Name := 'Compress Tobacco';
	ELSE
		Stage_Name := 'Comprimir Tabaco';
	END_IF
	
	IF qxClamp = FALSE THEN
		qxClamp:=TRUE;
		ClampTimer.IN:=TRUE;
		ClampTimer.PT:=Clamp_Security_Time;

	END_IF
	
	//IF Compress.Stage1Executed = FALSE THEN

	Compress._compress_tobacco(Enable:=TRUE);
	Compress.HomeExecuted:=FALSE;	
	
	IF Compress.axis_ready THEN	//Compress.Stage1Executed := FALSE;
		StateNext := 129;
		after_debug_state:=135;
		Compress._compress_tobacco(Enable:=FALSE);
		
		
		IF language.english THEN
			Stage_Name := 'Compress Tobacco done';
		ELSE
			Stage_Name := 'Comprimir tabaco concluído';
		END_IF
		
	END_IF
	//END_IF

131: //after_each_debug
	IF NOT ixStartButton AND NOT ixStart_Button_Machine THEN
	
		statenext:=after_debug_state;
	END_IF
135://stage2
	
	IF language.english THEN
		Stage_Name := concat('Shield-Pusher Stage ',INT_TO_STRING(stage_sh_push));
	ELSE
		Stage_Name := concat('Empurrador-proteção Estágio',INT_TO_STRING(stage_sh_push));
	END_IF
	
	Pusher.HomeExecuted:=FALSE;
	Shield.HomeExecuted:=FALSE;
		
	Pusher._absolute_move(Enable:=TRUE,Stage:=stage_sh_push);
	Shield._absolute_move(Enable:=TRUE,Stage:=stage_sh_push);
	IF pusher.axis_ready AND shield.axis_ready THEN	
		Statenext:= 129;
		IF stage_sh_push =6 THEN
			after_debug_state := 150;
			stage_sh_push:=0;
		ELSE
			after_debug_state := 135;
		END_IF
		Pusher._absolute_move(Enable:=FALSE,Stage:=stage_sh_push);
		Shield._absolute_move(Enable:=FALSE,Stage:=stage_sh_push);
		stage_sh_push:=stage_sh_push+1;
		
		IF language.english THEN
			Stage_Name:=concat(Stage_Name,' done');
		ELSE
			Stage_Name:=concat(Stage_Name,' concluído');
		END_IF
	END_IF	
	


150: //stage 5
	IF language.english THEN
		Stage_Name := 'Retract all';
	ELSE
		Stage_Name := 'Retrair tudo';
	END_IF
	//IF 	Shield._retract(Enable:=TRUE) AND Pusher._retract(Enable:=TRUE) AND Compress._retract(Enable:=TRRUE) THEN
	Pusher._Retract(enable:=TRUE);
	Shield._retract(enable:=TRUE);
	Compress._retract(enable:=TRUE);

	IF Compress.axis_ready AND Shield.Axis_ready AND Pusher.axis_ready THEN
		Pusher._Retract(enable:=FALSE);
		Shield._retract(enable:=FALSE);
		Compress._retract(enable:=FALSE);
		Statenext:=290;
		
		IF language.english THEN
			Stage_Name := 'Retract All Done';
		ELSE
			Stage_Name := 'Retrair tudo concluído';
		END_IF
	END_IF	

290:
	product_count:=product_count+1;
	statenext:=300;


300: //end
	
	Pusher.HomeExecuted:= TRUE;
	Shield.HomeExecuted:=TRUE;
	Compress.HomeExecuted:=TRUE;
	statenext:= 115;

	
1000: // overtorque
	
	//StartLoad := FALSE;
	
	tickcounter:=0;
	
	qxclamp:=FALSE;
	ClampTimer.IN:=FALSE;
	ClampTimer.PT:=Clamp_Security_Time;
	
	IF Pusher.PusherServo.xstopped AND Shield.ShieldServo.xstopped AND Compress.CompressServo.xstopped THEN
		Pusher._Reset();
		Shield._Reset();
		Compress._Reset();
		Statenext:=1005;
	END_IF

1005:
	
	IF tickcounter >1000 THEN
		statenext:=2000;
		tickcounter:=0;
	ELSE
		tickcounter:=tickcounter+1;
	END_IF

	
2000: // estop //overtorque
	
	tickcounter:= tickcounter+1;
	IF	tickcounter = 100 THEN
		tickcounter:=0;
		
		statenext:=15;
		overtorque_alarm:=FALSE;
	END_IF

2001: //guard
	tickcounter:= tickcounter+1;
	IF	tickcounter = 100 THEN
		tickcounter:=0;
		
		statenext:= 40;
		
	END_IF

2010: // clamp alarm
	
	tickcounter:= tickcounter+1;

	
	IF clamp_alarm THEN
		
		IF	tickcounter = 3000 THEN
			tickcounter:=0;
			statenext:=100;
			Clamp_Cooling := FALSE;
			Clamp_Alarm := FALSE;
		ELSE
			Clamp_Cooling := TRUE;
			
			IF Pusher.PusherServo.xstopped AND Shield.ShieldServo.xstopped AND Compress.CompressServo.xstopped THEN
				Pusher._Reset();
				Shield._Reset();
				Compress._Reset();
			END_IF
		END_IF
	END_IF 



2015://stop button
	tickcounter:= tickcounter+1;
	IF	tickcounter = 100 THEN
		tickcounter:=0;
		statenext:=100;
		
	ELSIF Pusher.PusherServo.xstopped AND Shield.ShieldServo.xstopped AND Compress.CompressServo.xstopped THEN
		Pusher._Reset();
		Shield._Reset();
		Compress._Reset();
		
	END_IF

2020: //force home

	IF shield.ShieldServo.xHalted AND pusher.pusherservo.xHalted AND compress.compressservo.xhalted THEN
		Pusher._soft_Reset();
		Shield._soft_Reset();
		Compress._soft_Reset();
		IF compress.offsetExecuted AND shield.Offsetexecuted AND pusher.offsetexecuted THEN
			statenext:=200;
		ELSE

			statenext:=210;
		END_IF
	END_IF

2030: //compress setting
	IF shield.ShieldServo.xHalted AND pusher.pusherservo.xHalted AND compress.compressservo.xhalted THEN
		Pusher._soft_Reset();
		Shield._soft_Reset();
		Compress._soft_Reset();
		
		
		Compress.HomeExecuted:=FALSE;
		Shield.HomeExecuted:=FALSE;
		Pusher.HomeExecuted:=FALSE;
	
		Compress.OffsetExecuted:=FALSE;
		Shield.OffsetExecuted:=FALSE;
		Pusher.OffsetExecuted:=FALSE;
		
		reset_rec_old();
		
		IF NOT compress_settings.done AND yellow_visibility.maintenance THEN
			statenext:=230;
		ELSE
			statenext:=115;
			compress_settings.done:=FALSE;
		END_IF
	END_IF


	
	
200:

	IF language.english THEN
		Stage_Name := 'Going to Home Position';	
	ELSE
		Stage_Name := 'Indo para Posição Inicial';
	END_IF
	
	
	
	Pusher._force_home(enable:=TRUE);
	
	IF tickcounter > 100 THEN
		Shield._force_home(enable:=TRUE);
	ELSE
		tickcounter:=tickcounter+1;
	END_IF
			
	Compress._force_home(enable:=TRUE);
	
	
	IF Compress.axis_ready AND Pusher.axis_ready AND Shield.Axis_ready THEN
		tickcounter:=0;
		Pusher._force_home(enable:=FALSE);
		Shield._force_home(enable:=FALSE);
		Compress._force_home(enable:=FALSE);
		Statenext:=300;
		
	END_IF

210:
	Compress.HomeExecuted:=FALSE;
	Shield.HomeExecuted:=FALSE;
	Pusher.HomeExecuted:=FALSE;
	
	Compress.OffsetExecuted:=FALSE;
	Shield.OffsetExecuted:=FALSE;
	Pusher.OffsetExecuted:=FALSE;
	
	Shield.Shield_param:=recipe_screen;
	Compress.Compress_Param := recipe_screen;
	Pusher.Pusher_Param := recipe_screen;
	
	reset_rec_old();
	
	Statenext:=211;

211:

	IF language.english THEN
		Stage_Name := 'Going to Home Position';	
	ELSE
		Stage_Name := 'Indo para Posição Inicial';
	END_IF
	
	IF Pusher.HomeExecuted = FALSE THEN 
		Pusher._Home();
		
	END_IF
	
	IF Compress.HomeExecuted = FALSE THEN
		Compress._Home();
		
	END_IF
	
	IF shield.HomeExecuted = FALSE THEN
		IF tickcounter>100 THEN
			Shield._Home();
		ELSE
			tickcounter:=tickcounter+1;
		END_IF
	END_IF
	
	IF Compress.HomeExecuted AND Pusher.HomeExecuted AND Shield.HomeExecuted THEN
		StateNext := 212;
		tickcounter:=0;                
		
	END_IF
	

212:

	IF Compress.OffsetExecuted = FALSE THEN
		Compress.Offset(enable:=TRUE);
	END_IF
	
	IF Shield.OffsetExecuted = FALSE THEN
		Shield.Offset(enable:=TRUE);
	END_IF
	
	IF Pusher.OffsetExecuted = FALSE THEN
		Pusher.Offset(enable:=TRUE);
	END_IF
	
	IF Pusher.OffsetExecuted AND Shield.OffsetExecuted AND Compress.OffsetExecuted THEN
		Pusher.Offset(enable:=FALSE);
		Shield.Offset(enable:=FALSE);
		Compress.Offset(enable:=FALSE);
		rec_old:= shield.Shield_Param;
		statenext:=300;
	END_IF

230:
	Compress._manuel(TRUE);
	
	IF compress_settings.find THEN
		statenext:=235;
		compress_settings.old_distance:=compress.compressservo.fActualPosition;
		Compress._manuel(FALSE);	
	END_IF
	
	IF compress_settings.done OR NOT yellow_visibility.maintenance THEN
		statenext:=2030;
		Compress._manuel(FALSE);
		compress_settings.distance_vis:=FALSE;
		//compress_settings.done:=FALSE;
		Compress._Halt();
		Shield._Halt();
		Pusher._Halt();
		
	END_IF
	
235://here
	Compress._Home_without_resetting(TRUE);
	compress_settings.distance_vis:=FALSE;
	
	IF Compress.axis_ready THEN
		Compress_settings.distance := Compress_settings.old_distance - compress.compressservo.fActualPosition;
		StateNext:=230;
		compress_settings.distance_vis:=TRUE;
		Compress._Home_without_resetting(FALSE);
	END_IF
	
	IF compress_settings.done OR NOT yellow_visibility.maintenance THEN
		statenext:=2030;
		Compress._Home_without_resetting(FALSE);
		compress_settings.distance_vis:=FALSE;
		//compress_settings.done:=FALSE;
		Compress._Halt();
		Shield._Halt();
		Pusher._Halt();
		
		
	END_IF


	
END_CASE

Pusher._Update();
Shield._Update();
Compress._Update();
ClampTimer();

axis_offset_or_not();

//maintenance visibility and stop button light
start_lamp_control();

//Motor Overtorque
motor_overtorque();



//Toggole Clamp
funct_toggle_clamp();

//Home
funct_force_home();

//stop button
funct_stop();

//Clamp Err
funct_clamp_err();

//compress setting
funct_compress_setting();


//guard
funct_guard_open();


//estop
funct_e_stop();

//IF State <> StateNext THEN - step through the state machine if required
coder_debug();

METHOD _debug : BOOL
VAR_INPUT
	enable				:BOOL;
END_VAR
IF enable THEN
	
	IF Debug_Mode THEN
		Maintenance_Visibility := TRUE;
		qxStartButtonLamp:=TRUE;
		IF (ixStartButton OR Step_Next OR ixStart_Button_Machine) THEN
			IF Parameter_Violation = FALSE THEN
				
				Step_Next:=FALSE;
				
				_debug:=TRUE;
				
				Maintenance_Visibility := FALSE;
				qxStartButtonLamp:=FALSE;
			
				Shield.Shield_param:=recipe_screen;
				Compress.Compress_Param := recipe_screen;
				Pusher.Pusher_Param := recipe_screen;
			ELSE
				Step_Next:=FALSE;
			END_IF
		END_IF
	ELSE
		//StateNext:=130;
		_debug:=TRUE;
		Maintenance_Visibility := FALSE;
	END_IF
	
	
ELSE
	_debug:=FALSE;
END_IF
END_METHOD

METHOD axis_offset_or_not : BOOL
VAR_INPUT
END_VAR
	//rec_old:=Shield.Shield_Param;     //old values

	
	//Shield.Shield_param:=recipe_screen;         //new valuses
	//Compress.Compress_Param := recipe_screen;
	//Pusher.Pusher_Param := recipe_screen;
	
IF statenext<>127 AND statenext<> 212 THEN
	IF rec_old.other.Shield_Home_Offset <> recipe_screen.Other.Shield_Home_Offset THEN

		Shield.OffsetExecuted:=FALSE;
	END_IF
	
	IF rec_old.other.Pusher_Home_Offset <> recipe_screen.Other.Pusher_Home_Offset THEN
		Pusher.OffsetExecuted:=FALSE;
	END_IF
	
	IF rec_old.other.Compress_Home_Offset <> recipe_screen.Other.Compress_Home_Offset THEN
		Compress.OffsetExecuted:=FALSE;
	END_IF
END_IF
END_METHOD

METHOD coder_debug : BOOL
VAR_INPUT
END_VAR
IF singleStep AND statenext > 119 THEN
	//IF NOT SM_StepRequest THEN
	//	SM_StepRequest := TRUE; 
	//END_IF
	IF SM_StepRequest THEN
		SM_StepRequest := FALSE;
		State := StateNext;
	END_IF
ELSE
	State := StateNext;
END_IF
END_METHOD

METHOD funct_clamp_err : BOOL
VAR_INPUT
END_VAR
IF (Clamptimer.Q=TRUE) AND StateNext >= 100 AND StateNext <= 300 THEN 
	
	tickcounter:=0;
	//Message:='Clamp Overtime';
	qxClamp:=FALSE;

	
	ClampTimer.IN:=FALSE;
	ClampTimer.PT:=Clamp_Security_Time;
	
	Clamp_Alarm:=TRUE;
	
	Compress._mc_stop();
	Shield._mc_stop();
	Pusher._mc_stop();
	StateNext := 2010;

END_IF
END_METHOD

METHOD funct_compress_setting : BOOL
VAR_INPUT
END_VAR
IF compress_settings.button AND StateNext >= 115 AND StateNext <= 300 THEN
	compress_settings.button:=FALSE;
	
	IF statenext < 230 OR statenext >250 THEN
		StateNext := 2030;
		tickcounter:=0;
	
		compress_settings.done:=FALSE;
	
	
		qxclamp:=FALSE;
		ClampTimer.IN:=FALSE;
		ClampTimer.PT:=Clamp_Security_Time;
	
		shield._Halt();
		pusher._Halt();
		compress._Halt();
	END_IF
	
ELSE
	compress_settings.button:=FALSE;
END_IF
END_METHOD

METHOD funct_e_stop : BOOL
VAR_INPUT
END_VAR
IF (NOT ixCabinetE_StopButtonOkay) AND StateNext >= 30 AND StateNext <= 300 THEN 
	
	tickcounter:=0;
	
	//Message:='E-stop Pressed';
	
	qxclamp:=FALSE;
	ClampTimer.IN:=FALSE;
	ClampTimer.PT:=Clamp_Security_Time;
	

	
	//IF Compress.CompressServo.xStopped AND Shield.ShieldServo.xStopped AND Pusher.PusherServo.xStopped THEN
	StateNext := 2000;
	Pusher._Reset();
	Shield._Reset();
	Compress._Reset();
	//END_IF
END_IF
END_METHOD

METHOD funct_force_home : BOOL
VAR_INPUT
END_VAR
IF (Force_Home) AND StateNext >= 115 AND StateNext <= 300 THEN 
	Force_Home:=FALSE;
	
	IF statenext < 200 OR statenext >220 THEN
		StateNext := 2020;
		tickcounter:=0;
	
	
	
	
		qxclamp:=FALSE;
		ClampTimer.IN:=FALSE;
		ClampTimer.PT:=Clamp_Security_Time;
	
		shield._Halt();
		pusher._Halt();
		compress._Halt();
	END_IF

END_IF
END_METHOD

METHOD funct_guard_open : BOOL
VAR_INPUT
END_VAR
IF (NOT ixGuardRelayOkay) AND StateNext >= 50 AND StateNext <= 300 THEN 
	
	StateNext := 2001;
	tickcounter:=0;
	
	//Message:='Guard Open';
	
	qxclamp:=FALSE;
	ClampTimer.IN:=FALSE;
	ClampTimer.PT:=Clamp_Security_Time;
	
	IF Pusher.HomeExecuted= FALSE OR Shield.HomeExecuted = FALSE OR Compress.HomeExecuted = FALSE THEN
		Pusher._Reset();
		Shield._Reset();
		Compress._Reset();
	ELSE
		Pusher._Reset_Medium();
		Shield._Reset_Medium();
		Compress._Reset_Medium();
	END_IF
END_IF
END_METHOD

METHOD funct_stop : BOOL
VAR_INPUT
END_VAR
IF NOT ixstop_button AND (Statenext<>151) AND StateNext >= 100 AND StateNext <= 300 THEN
	//	state_old:=statenext;
	//	statenext:= 151;
	tickcounter:=0;
	//Message:='Clamp Overtime';
	qxClamp:=FALSE;

	
	ClampTimer.IN:=FALSE;
	ClampTimer.PT:=Clamp_Security_Time;
	
	
	
	Compress._mc_stop();
	Shield._mc_stop();
	Pusher._mc_stop();
	StateNext := 2015;
	
	
END_IF
END_METHOD

METHOD funct_toggle_clamp : BOOL
VAR_INPUT
END_VAR
IF StateNext >= 115 AND StateNext <= 300 AND Toggle_Clamp THEN
	Toggle_Clamp := FALSE;
	IF qxClamp = FALSE THEN
		
		qxClamp:=TRUE;
		ClampTimer.IN:=TRUE;
		ClampTimer.PT:=Clamp_Security_Time;

	ELSE
		
		qxClamp:=FALSE;
		ClampTimer.IN:=FALSE;
		ClampTimer.PT:=Clamp_Security_Time;
		
	END_IF
	
	
END_IF
END_METHOD

METHOD motor_overtorque : BOOL
VAR
	torque_lim			:LREAL;
	current_torque_shield		:LREAL;
	current_torque_compress		:LREAL;
	current_torque_pusher		:LREAL;
	
END_VAR
IF StateNext >= 110 AND StateNext <= 300  THEN					// machine is running
	
	torque_lim:=limits_screen.max_torque;
	//torque_lim:=2000;
	
	current_torque_shield:=ibshieldservotorque;
	current_torque_pusher:=ibpusherservotorque;
	current_torque_compress:=ibcompressservotorque;
	
	IF current_torque_compress  > torque_lim OR current_torque_compress  < (-1*torque_lim) THEN					
		//Message := WSTRING_TO_STRING("Tobacco Compress Servo over-torque");
		StateNext := 1000;
		tickcounter:=0;
		overtorque_alarm:= TRUE;

		compress._mc_stop();
		shield._mc_stop();
		pusher._mc_stop();	
	END_IF
	
	IF current_torque_pusher  > torque_lim OR current_torque_pusher  < (-1*torque_lim) THEN						
		//Message := WSTRING_TO_STRING("Rod Pusher Servo over-torque");
		StateNext := 1000;
		tickcounter:=0;
		overtorque_alarm:= TRUE;
		
		compress._mc_stop();
		shield._mc_stop();
		pusher._mc_stop();	
			
	END_IF
	
	IF current_torque_shield  > torque_lim OR current_torque_shield  < (-1*torque_lim) THEN						
		//Message := WSTRING_TO_STRING("Rod Shield Servo over-torque");
		StateNext := 1000;
		tickcounter:=0;
		overtorque_alarm:= TRUE;

		compress._mc_stop();
		shield._mc_stop();
		pusher._mc_stop();		
	END_IF
END_IF
END_METHOD

METHOD reset_rec_old : BOOL
VAR_INPUT
END_VAR
rec_old:=empty_recipe;
END_METHOD

METHOD start_lamp_control : BOOL
VAR_INPUT
END_VAR
//IF 	StateNext <> 115 AND 
//	StateNext <> 127 THEN
//	qxStartButtonLamp:=FALSE;
//END_IF

IF 	StateNext <> 115 AND StateNext <> 127 AND StateNext <> 129 THEN
	qxStartButtonLamp:=FALSE;
	Maintenance_Visibility := FALSE;
END_IF
END_METHOD

METHOD StopClampTimer
VAR_INPUT
END_VAR
ClampTimer.IN:=FALSE;
ClampTimer.PT:= Clamp_Security_Time;
END_METHOD

END_PROGRAM

// ---- Classes/Pusher/FB_Pusher.TcPOU
FUNCTION_BLOCK FB_Pusher
VAR_INPUT
END_VAR
VAR_OUTPUT
	axis_ready				:BOOL:=FALSE;
END_VAR
VAR

PusherServo        			:FB_AxisControl;

_Pusher_param				:recipe;



ToolPositioningSpeed	: LREAL := 20;
ToolPositioningAccel	: LREAL := 100;
ToolPositioningJerk		: LREAL := 1000;
ToolHomingSpeed			: LREAL := 2;

PusherServoEnable			:BOOL;
PusherServoEnabled			:BOOL;

_ExecutedHome				:BOOL:=FALSE;
_ExecutedStage2				:BOOL:=FALSE;
_ExecutedStage4				:BOOL:=FALSE;
_ExecutedStage5				:BOOL:=FALSE;
_ExecutedOffset				:BOOL:=FALSE;
_ExecutedTamp				:BOOL:=FALSE;

tickcounter_pusher: 		INT :=0;
State: 						INT:= 0;
StateNext: 					INT:= 0;

pusher_old_position			:LREAL;




END_VAR

METHOD _absolute_move : BOOL
VAR_INPUT
	Enable				:BOOL;
	Stage				:INT;
END_VAR
IF Enable AND NOT axis_ready THEN
	CASE State OF
	
	0:	
		
		PusherServo.fPosition:= _Pusher_Param.Pusher.Distance[Stage];
		PusherServo.fVelocity:= _Pusher_Param.Pusher.Speed[Stage]; //mm/s
	
		IF stage = 6 THEN
			_Pusher_Param.Clamp.Release_Instance := _Pusher_Param.Clamp.Release_Instance - _Pusher_Param.Pusher.Distance[5];
		
			IF _Pusher_Param.Clamp.Release_Instance <= 0 THEN
				IF qxClamp = TRUE THEN
					qxClamp:=FALSE;
					PRG_Machine.StopClampTimer();
	
				END_IF
			END_IF
	
			pusher_old_position:= PusherServo.fActualPosition;
		END_IF 
		
		PusherServo.xMoveA:=TRUE;
	
	
		StateNext:=5;
	5:	
		IF PusherServo.xInPosition = TRUE THEN
		
			PusherServo.xMoveA := FALSE;
			StateNext:=0;
			axis_ready:=TRUE;
		
			IF qxClamp = TRUE AND Stage = 6 THEN
				qxClamp:=FALSE;
		
				PRG_Machine.StopClampTimer();
	
			END_IF
		END_IF
		
		IF (PusherServo.fActualPosition-pusher_old_position) >= (_Pusher_Param.Clamp.Release_Instance) AND Stage = 6 THEN
			IF qxClamp = TRUE THEN
				qxClamp:=FALSE;
		
				PRG_Machine.StopClampTimer();
	
			END_IF
		END_IF


	END_CASE

	State:=StateNext;
ELSIF NOT enable THEN 
	axis_ready:=FALSE;
	PusherServo.xMoveA := FALSE;
	state:=0;
	statenext:=0;
END_IF
END_METHOD

METHOD _Enable 
VAR_INPUT
END_VAR

PusherServoEnable := TRUE;
END_METHOD

METHOD _force_home  : BOOL
VAR_INPUT
	Enable				:BOOL;
	
END_VAR
IF enable AND NOT axis_ready THEN
	CASE State OF
	
	0:	
	
		PusherServo.fPosition:= 0;
		PusherServo.fVelocity:= 10; //mm/s
	
		PusherServo.xMoveA:=TRUE;
		StateNext:=5;
	5:	
		IF PusherServo.xInPosition = TRUE THEN
		
			PusherServo.xMoveA := FALSE;
			StateNext:=0;
			axis_ready:=TRUE;
		
		END_IF


	END_CASE

	State:=StateNext;
ELSIF NOT enable THEN
	axis_ready:=FALSE;
	PusherServo.xMoveA := FALSE;
	state:=0;
	statenext:=0;
END_IF
END_METHOD

METHOD _Halt : BOOL
VAR_INPUT
END_VAR
PusherServo.xHalt:=TRUE;
END_METHOD

METHOD _Halt_false : BOOL
VAR_INPUT
END_VAR
PusherServo.xHalt:=FALSE;
END_METHOD

METHOD _Home 
VAR_INPUT
	
END_VAR


VAR


END_VAR

VAR_OUTPUT
	
END_VAR


CASE State OF //you are here



0:	
	_ExecutedHome := FALSE;
	PusherServo.fVelocity := ToolPositioningSpeed;
	PusherServo.fAxisAcceleration := ToolPositioningAccel;
	PusherServo.fAxisDeceleration := ToolPositioningAccel;
	PusherServo.fAxisJerk := ToolPositioningJerk;

	IF ixPusherHomeSwitch THEN
		PusherServo.xPositiveDirection := FALSE;
		IF  tickcounter_pusher < 10 THEN
			tickcounter_pusher := tickcounter_pusher + 1;  // can be put in onditional
		
		ELSE
		//IF tickcounter_compress >= 10 THEN
			PusherServo.xMoveV := TRUE;
		END_IF
	ELSE
	
		//CompressServo.xHalt := NOT CompressServo.xHalt;
		PusherServo.xMoveV := FALSE;
		//CompressServo.xHalt := NOT CompressServo.xHalt;
		PusherServo.xHalt := TRUE;
		IF PusherServo.xHalted THEN
			tickcounter_pusher:=0;
			StateNext := 5;
		END_IF
	
	END_IF
	
5:
	
	PusherServo.xHalt := FALSE;
	tickcounter_Pusher := tickcounter_Pusher + 1;
	IF tickcounter_Pusher >= 10 THEN
		tickcounter_Pusher := 0;
		StateNext := 10;
	END_IF
	
10:
	PusherServo.fVelocity := ToolHomingSpeed;
	
	IF NOT ixPusherHomeSwitch THEN
		PusherServo.xPositiveDirection := TRUE;
		IF tickcounter_Pusher < 10 THEN
			tickcounter_Pusher := tickcounter_Pusher + 1;
		ELSE
		//IF tickcounter >= 10 THEN
			PusherServo.xMoveV := TRUE;
		END_IF
	ELSE
		PusherServo.xMoveV := FALSE;
		PusherServo.xHalt := TRUE;
		IF PusherServo.xHalted AND PusherServo.fstandstill THEN
			tickcounter_Pusher := 0;
			StateNext := 15;
		END_IF
	END_IF

15:
	
	PusherServo.xHalt := FALSE;
	tickcounter_Pusher := tickcounter_Pusher + 1;
	IF tickcounter_Pusher >= 25 THEN
		tickcounter_Pusher := 0;
		StateNext := 20;
		//Executed := TRUE;
	END_IF
20:
	PusherServo.fHomeOffset := 0;
	PusherServo.xZero := TRUE;
	StateNext := 25;	
	
25:
	IF PusherServo.xZeroed THEN
		PusherServo.xZero := FALSE;
		_ExecutedHome := TRUE;
		StateNext := 0;
	END_IF
	

END_CASE

State := StateNext;
END_METHOD

METHOD _mc_stop : BOOL
VAR_INPUT
END_VAR
PusherServo.xStop:=TRUE;
END_METHOD

METHOD _Reset
VAR_INPUT
END_VAR
	tickcounter_Pusher:=0;
	PusherServoEnable := FALSE;
	PusherServo.xZero := FALSE;
	PusherServo.xMoveV := FALSE;
	PusherServo.xMoveA := FALSE;
	PusherServo.xHalt := FALSE;
	PusherServo.GearIn := FALSE;
	PusherServo.xStop:=FALSE;
	state:=0;
	statenext:=0;
	
	
	axis_ready:=FALSE;
	_ExecutedHome:=FALSE;
	_ExecutedOffset:=FALSE;
	PRG_Machine.reset_rec_old();
	PRG_Machine._debug(enable:=FALSE);
END_METHOD

METHOD _Reset_medium
VAR_INPUT
END_VAR
	tickcounter_Pusher:=0;
	PusherServoEnable := FALSE;
	PusherServo.xZero := FALSE;
	PusherServo.xMoveV := FALSE;
	PusherServo.xMoveA := FALSE;
	PusherServo.xHalt := FALSE;
	PusherServo.GearIn := FALSE;
	PusherServo.xStop:=FALSE;
	state:=0;
	statenext:=0;
	
	
	axis_ready:=FALSE;
	PRG_Machine._debug(enable:=FALSE);
END_METHOD

METHOD _retract  : BOOL
VAR_INPUT
	Enable				:BOOL;
	
END_VAR
IF enable AND NOT axis_ready THEN
	CASE State OF
	
	0:	
	
		PusherServo.fPosition:= 0;
		PusherServo.fVelocity:= _Pusher_Param.Pusher.Retract_Speed; //mm/s
	
		PusherServo.xMoveA:=TRUE;
		StateNext:=5;
	5:	
		IF PusherServo.xInPosition = TRUE THEN
		
			PusherServo.xMoveA := FALSE;
			StateNext:=0;
			axis_ready:=TRUE;
		
		END_IF


	END_CASE

	State:=StateNext;
ELSIF NOT enable THEN
	axis_ready:=FALSE;
	PusherServo.xMoveA := FALSE;
	state:=0;
	
END_IF
END_METHOD

METHOD _Soft_Reset
VAR_INPUT
END_VAR

tickcounter_Pusher:=0;
PusherServo.xZero := FALSE;
PusherServo.xMoveV := FALSE;
PusherServo.xMoveA := FALSE;
PusherServo.xHalt := FALSE;
PusherServo.GearIn := FALSE;
PusherServo.xStop:=FALSE;
state:=0;
statenext:=0;

axis_ready:=FALSE;
PRG_Machine._debug(enable:=FALSE);
END_METHOD

METHOD _Update
VAR_INPUT
END_VAR
PusherServo(
	xEnable:= PusherServoEnable, 
	xZero:= , 
	xMoveR:= , 
	xMoveA:= , 
	xMoveV:= , 
	xPositiveDirection:= , 
	fDistance:= , 
	fPosition:= , 
	fVelocity:= , 
	xStop:= , 
	xHome:= , 
	xHomeFlag:= , 
	homePosition:=0,
	fActualPosition=> , 
	fActualVelocity=> , 
	fActModuloPos=> , 
	xEnabled=> PusherServoEnabled, 
	xMoveComplete=> , 
	xInPosition=> , 
	xAtSpeed=> , 
	xStopped=> , 
	xHomed=> ,
	errorID=> PusherServoErrorID, 
	Axis:= PusherAxis );
END_METHOD

PROPERTY HomeExecuted : BOOL
GET
HomeExecuted := _ExecutedHome;
END_GET
SET
_ExecutedHome := HomeExecuted;
END_SET
END_PROPERTY

METHOD Offset
VAR_INPUT
	Enable				:BOOL;
END_VAR

IF enable AND NOT axis_ready THEN	
	CASE State OF
	0:	
		_ExecutedOffset:=FALSE;
		PusherServo.fPosition:= _Pusher_Param.Other.Pusher_Home_Offset-PRG_Machine.rec_old.other.pusher_home_offset;
		PusherServo.fVelocity:= 20; //mm/s
	
		IF PusherServo.fPosition<>0 THEN
			PusherServo.xMoveA:=TRUE;
			StateNext:=5;
		ELSE
			_ExecutedOffset:=TRUE;
		END_IF
	
		//StateNext:=5;
	5:	
		IF PusherServo.xInPosition = TRUE AND PusherServo.fstandstill THEN
			
			PusherServo.xMoveA := FALSE;
			StateNext:=7;
			//_ExecutedOffset:=TRUE;
		
		END_IF
	7:
		tickcounter_pusher:=tickcounter_pusher+1;
		IF tickcounter_Pusher >= 25 THEN
			tickcounter_Pusher := 0;
			StateNext := 10;
			//Executed := TRUE;
		END_IF	
	
	10:
	
		PusherServo.fHomeOffset := 0;
		pusherServo.xZero := TRUE;
		StateNext := 15;	
	
	15:
		IF pusherServo.xZeroed THEN
			pusherServo.xZero := FALSE;
			_ExecutedOffset:=TRUE;
			axis_ready:=TRUE;
			StateNext := 0;
		END_IF

	END_CASE

	State:=StateNext;
	
ELSIF NOT enable THEN 
	axis_ready:=FALSE;
	pusherServo.xZero := FALSE;
	StateNext := 0;
END_IF
END_METHOD

PROPERTY OffsetExecuted : BOOL
GET
OffsetExecuted := _ExecutedOffset;
END_GET
SET
_ExecutedOffset := OffsetExecuted;
END_SET
END_PROPERTY

PROPERTY Pusher_Param : recipe
GET
Pusher_param := _Pusher_Param;
END_GET
SET
_Pusher_param := Pusher_Param;
END_SET
END_PROPERTY

PROPERTY Stage2Executed : BOOL
GET
Stage2Executed := _ExecutedStage2;
END_GET
SET
_ExecutedStage2 := Stage2Executed;
END_SET
END_PROPERTY

PROPERTY Stage4Executed : BOOL
GET
Stage4Executed := _ExecutedStage4;
END_GET
SET
_ExecutedStage4 := Stage4Executed;
END_SET
END_PROPERTY

PROPERTY Stage5Executed : BOOL
GET
Stage5Executed := _ExecutedStage5;
END_GET
SET
_ExecutedStage5 := Stage5Executed;
END_SET
END_PROPERTY

PROPERTY TampExecuted : BOOL
GET
TampExecuted := _ExecutedTamp;
END_GET
SET
_ExecutedTamp := TampExecuted;
END_SET
END_PROPERTY

END_FUNCTION_BLOCK

// ---- POUs/FB_AxisControl.TcPOU
FUNCTION_BLOCK FB_AxisControl
VAR_INPUT
	xEnable: BOOL;
	xZero: BOOL;
	xMoveR: BOOL;
	xMoveA: BOOL;
	xMoveV: BOOL;
	xPositiveDirection: BOOL;
	fDistance: LREAL;
	fPosition: LREAL;
	fVelocity: LREAL;
	xStop: BOOL;
	xHome: BOOL;
	xHomeFlag: BOOL;
	xHalt: BOOL;
	xTimerInput: BOOL;
	timerPT: TIME;
	HomePosition: LREAL;
	fAxisAcceleration: LREAL;
	fAxisDeceleration: LREAL;
	fAxisJerk: LREAL;
	MasterAxis: AXIS_REF;
	GearIn: BOOL;
	Gear_out: BOOL;
	GearRatio: LREAL;
	EnableSoE_ReadPosition: BOOL;
	EnableSoE_ReadTorque: BOOL;
	EnableSoE_ReadFollowingError: BOOL;
	fHomeOffset: LREAL;
END_VAR
VAR_OUTPUT
	gear_out_busy	:BOOL;
	fActualPosition: LREAL;
	fActualVelocity: LREAL;
	fActModuloPos: LREAL;
	fActPosition: DINT;
	fActFollowingError: DINT;
	fActualTorque: LREAL;
	xEnabled: BOOL;
	xMoveComplete: BOOL;
	xInPosition: BOOL;
	xAtSpeed: BOOL;
	xStopped: BOOL;
	xHomed: BOOL;
	xHalted: BOOL;
	errorID: UDINT;
	xAxisHomed: BOOL;
	xZeroed: BOOL;
	timerET: TIME;
	timerQOutput: BOOL;
	InGear: BOOL;
	xServoError: BOOL;
	iErrorID: UDINT;
	fstandstill: BOOL;
END_VAR
VAR
	mcPower: MC_Power;
	mcReset: MC_Reset;
	mcMoveRelative: MC_MoveRelative;
	mcSetPosition: MC_SetPosition;
	mcMoveAbsolute: MC_MoveAbsolute;
	mcReadStatus: MC_ReadStatus;
	mcMoveVelocity: MC_MoveVelocity;
	mcStop: MC_Stop;
	mcHome: MC_Home;
	mcHalt: MC_Halt;
	timerOn: TON;

	mcGearInDyn: MC_GearInDyn;
	mcGearOut: MC_GearOut;
	
	EnReadPosition: BOOL;
	EnReadTorque: BOOL;
	EnReadFollowingError: BOOL;
	
END_VAR
VAR_IN_OUT
	Axis: AXIS_REF;
	//MasterAxis : AXIS_REF;
END_VAR

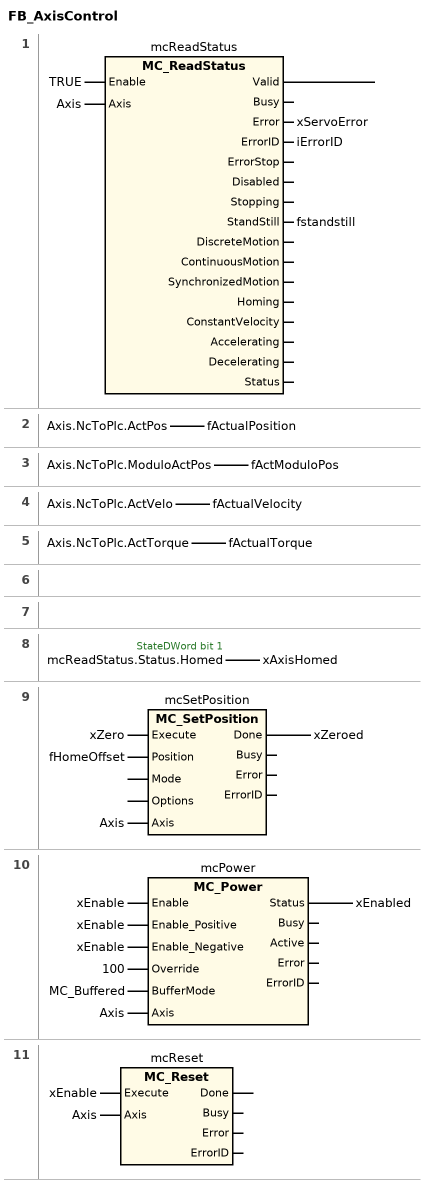
// NETWORK 1
mcReadStatus(
    Enable := TRUE,
    Axis := Axis,
    Error => xServoError,
    ErrorID => iErrorID,
    StandStill => fstandstill); // MC_ReadStatus

// NETWORK 2
fActualPosition := Axis.NcToPlc.ActPos;

// NETWORK 3
fActModuloPos := Axis.NcToPlc.ModuloActPos;

// NETWORK 4
fActualVelocity := Axis.NcToPlc.ActVelo;

// NETWORK 5
fActualTorque := Axis.NcToPlc.ActTorque;

// NETWORK 6

// NETWORK 7

// NETWORK 8
//   mcReadStatus.Status.Homed: StateDWord bit 1
xAxisHomed := mcReadStatus.Status.Homed;

// NETWORK 9
mcSetPosition(Execute := xZero, Position := fHomeOffset, Axis := Axis); // MC_SetPosition
xZeroed := mcSetPosition.Done;

// NETWORK 10
mcPower(
    Enable := xEnable,
    Enable_Positive := xEnable,
    Enable_Negative := xEnable,
    Override := 100,
    BufferMode := MC_Buffered,
    Axis := Axis); // MC_Power
xEnabled := mcPower.Status;

// NETWORK 11
mcReset(Execute := xEnable, Axis := Axis); // MC_Reset

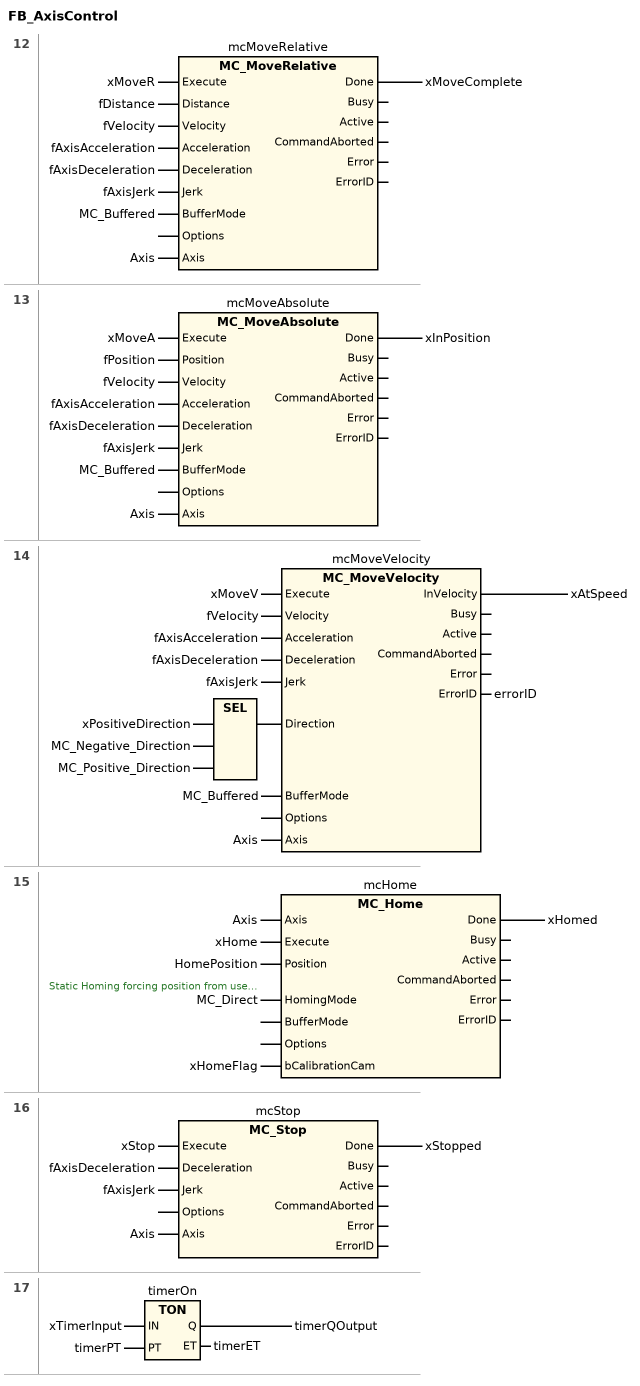
// NETWORK 12
mcMoveRelative(
    Execute := xMoveR,
    Distance := fDistance,
    Velocity := fVelocity,
    Acceleration := fAxisAcceleration,
    Deceleration := fAxisDeceleration,
    Jerk := fAxisJerk,
    BufferMode := MC_Buffered,
    Axis := Axis); // MC_MoveRelative
xMoveComplete := mcMoveRelative.Done;

// NETWORK 13
mcMoveAbsolute(
    Execute := xMoveA,
    Position := fPosition,
    Velocity := fVelocity,
    Acceleration := fAxisAcceleration,
    Deceleration := fAxisDeceleration,
    Jerk := fAxisJerk,
    BufferMode := MC_Buffered,
    Axis := Axis); // MC_MoveAbsolute
xInPosition := mcMoveAbsolute.Done;

// NETWORK 14
mcMoveVelocity(
    Execute := xMoveV,
    Velocity := fVelocity,
    Acceleration := fAxisAcceleration,
    Deceleration := fAxisDeceleration,
    Jerk := fAxisJerk,
    Direction := SEL(xPositiveDirection, MC_Negative_Direction, MC_Positive_Direction),
    BufferMode := MC_Buffered,
    Axis := Axis,
    ErrorID => errorID); // MC_MoveVelocity
xAtSpeed := mcMoveVelocity.InVelocity;

// NETWORK 15
//   MC_Direct: Static Homing forcing position from user reference
mcHome(
    Axis := Axis,
    Execute := xHome,
    Position := HomePosition,
    HomingMode := MC_Direct,
    bCalibrationCam := xHomeFlag); // MC_Home
xHomed := mcHome.Done;

// NETWORK 16
mcStop(Execute := xStop, Deceleration := fAxisDeceleration, Jerk := fAxisJerk, Axis := Axis); // MC_Stop
xStopped := mcStop.Done;

// NETWORK 17
timerOn(IN := xTimerInput, PT := timerPT, ET => timerET); // TON
timerQOutput := timerOn.Q;

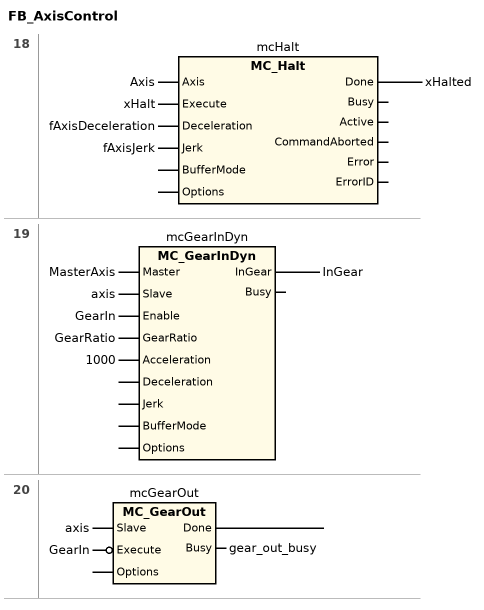
// NETWORK 18
mcHalt(Axis := Axis, Execute := xHalt, Deceleration := fAxisDeceleration, Jerk := fAxisJerk); // MC_Halt
xHalted := mcHalt.Done;

// NETWORK 19
mcGearInDyn(
    Master := MasterAxis,
    Slave := axis,
    Enable := GearIn,
    GearRatio := GearRatio,
    Acceleration := 1000); // MC_GearInDyn
InGear := mcGearInDyn.InGear;

// NETWORK 20
mcGearOut(Slave := axis, Execute := NOT GearIn, Busy => gear_out_busy); // MC_GearOut

END_FUNCTION_BLOCK

// ---- Classes/Compress/FB_Compress.TcPOU
FUNCTION_BLOCK FB_Compress
VAR_INPUT
END_VAR
VAR_OUTPUT
	axis_ready					:BOOL:=FALSE;
END_VAR
VAR

CompressServo: 				FB_AxisControl;

_Compress_param				:recipe;


ToolPositioningSpeed	: LREAL := 20;
ToolPositioningAccel	: LREAL := 100;
ToolPositioningJerk		: LREAL := 1000;
ToolHomingSpeed			: LREAL := 2;

CompressServoEnable:		BOOL;
CompressServoEnabled:		BOOL;

_ExecutedHome:				BOOL:=FALSE;
_ExecutedStage1:			BOOL:=FALSE;
_ExecutedStage5:			BOOL:=FALSE;
_ExecutedOffset:			BOOL:=FALSE;				

tickcounter_compress: 		INT :=0;
State: 						INT:= 0;
StateNext: 					INT:= 0;
			
	

END_VAR

METHOD _compress_tobacco 
VAR_INPUT
	Enable		:BOOL;
END_VAR
VAR

END_VAR
IF(Enable AND NOT axis_ready) THEN
	CASE State OF
	
	0:	
		//_ExecutedStage1:=FALSE;
		CompressServo.fPosition:= _Compress_Param.Compress.Initial_Distance;
		CompressServo.fVelocity:= _Compress_Param.Compress.Initial_Speed;
		CompressServo.xMoveA:=TRUE;
		StateNext:=5;
	5:	
		IF CompressServo.xInPosition = TRUE THEN
		
			CompressServo.xMoveA := FALSE;
			StateNext:=10;
		END_IF

	10:
		CompressServo.fVelocity:= _Compress_Param.Compress.Initial_Speed;
		CompressServo.fPosition:= _Compress_Param.Compress.Relax_Distance;
		CompressServo.xMoveA := TRUE;
		StateNext:=15;
	
	15:
		IF CompressServo.xInPosition = TRUE THEN
		
			CompressServo.xMoveA := FALSE;
			StateNext:=0;
			//_ExecutedStage1:=TRUE;
			axis_ready:=TRUE;
		END_IF

	

	END_CASE

	State:=StateNext;
	
ELSIF NOT enable THEN
	
	axis_ready:=FALSE;
	CompressServo.xMoveA := FALSE;
	StateNext:=0;
	state:=0;
	
END_IF
END_METHOD

METHOD _Enable 
VAR_INPUT
END_VAR

CompressServoEnable := TRUE;
END_METHOD

METHOD _force_home : BOOL
VAR_INPUT
	enable			:BOOL;
END_VAR
IF enable AND NOT axis_ready THEN
	CASE State OF
	
	0:	
	
